DATA_BLOCK "ASW_GraphicData"	// DB 80
TITLE = COPYRIGHT:    (C) 2003  BUHLER AG, CH-9240 UZWIL, SWITZERLAND
//
//PRODUCT:      GP_GCS7
//
//TITLE:        
//
//------------------------------------------------------------------------------------------------------
//
//IDENT:               AUTHOR:         DEPT:                 DATE:
//
//DB80.1A            CE                    FU53                    03.03.2003
//
//------------------------------------------------------------------------------------------------------
//
//PURPOSE:      MANUAL : see [MxxMAN]
//
//RESTRICTIONS: 
//------------------------------------------------------------------------------------------------------
//
//
//
//
AUTHOR : CE
FAMILY : GEN
VERSION : 0.0
  STRUCT
   spare0 : WORD ;
   Buttons : STRUCT
    Fault_F : UDT 1000;	//Fault_F1...Fault_F10
    Fault_SF : UDT 1000;	//Fault_SF1...Fault_SF10
    Active_F : UDT 1000;	//Active_F1...Active_F10
    Active_SF : UDT 1000;	//Active_SF1...Active_SF10
    Manual_F : UDT 1000;	//Manual_F1...Manual_F10
    Manual_SF : UDT 1000;	//Manual_SF1...Manual_SF10
   END_STRUCT ;
   spare14 : ARRAY  [14 .. 29 ] OF BYTE ;
   Way : STRUCT
    F01 : UDT 1001;	//F01L00 ... F01L09
    F02 : UDT 1001;	//F02L00 ... F02L09
    F03 : UDT 1001;	//F03L00 ... F03L09
    F04 : UDT 1001;	//F04L00 ... F04L09
    F05 : UDT 1001;	//F05L00 ... F05L09
    F06 : UDT 1001;	//F06L00 ... F06L09
    F07 : UDT 1001;	//F07L00 ... F07L09
    F08 : UDT 1001;	//F08L00 ... F08L09
    F09 : UDT 1001;	//F09L00 ... F09L09
    F10 : UDT 1001;	//F10L00 ... F10L09
    SF01 : UDT 1001;	//SF01L00 ... SF01L09
    SF02 : UDT 1001;	//SF02L00 ... SF02L09
    SF03 : UDT 1001;	//SF03L00 ... SF03L09
    SF04 : UDT 1001;	//SF04L00 ... SF04L09
    SF05 : UDT 1001;	//SF05L00 ... SF05L09
    SF06 : UDT 1001;	//SF06L00 ... SF06L09
    SF07 : UDT 1001;	//SF07L00 ... SF07L09
    SF08 : UDT 1001;	//SF08L00 ... SF08L09
    SF09 : UDT 1001;	//SF09L00 ... SF09L09
    SF10 : UDT 1001;	//SF10L00 ... SF10L09
   END_STRUCT ;
   Spare430 : ARRAY  [430 .. 499 ] OF BYTE ;
   General : STRUCT
    EmergencyStop : STRUCT
     SystemReset : BOOL ;	//Reset Emergency System
    END_STRUCT ;
    Horn : STRUCT
     Quit : ARRAY  [1 .. 16 ] OF //SwitchOff Horn 1..16
     BOOL ;
     Color : ARRAY  [1 .. 16 ] OF //Horn 1..16 is on
     BOOL ;
    END_STRUCT ;
    CycleTime : ARRAY  [1 .. 3 ] OF //Cycle Time Cycle 1..3
    STRUCT
     Minimal : INT ;	//Min. Cycle Time
     Actual : INT ;	//Act. Cycle Time
     Maximal : INT ;	//Max. Cycle Time
    END_STRUCT ;
    PCS : STRUCT
     PICNotOnline : BOOL ;	//ProcessControlSystem is not online
     Reserve : BOOL ;
    END_STRUCT ;
    Spare526 : STRUCT
     Reserve : ARRAY  [526 .. 549 ] OF BYTE ;
    END_STRUCT ;
   END_STRUCT ;
   UserPictureData : STRUCT
    F1 : STRUCT 	//User Data in Picture F1
     Binaer1 : STRUCT
      Bit0 : BOOL ;
      Bit01 : BOOL ;
      Bit02 : BOOL ;
     END_STRUCT ;
     Binaer2 : STRUCT
      Bit0 : BOOL ;
      Bit01 : BOOL ;
      Bit02 : BOOL ;
     END_STRUCT ;
     Binaer3 : STRUCT
      Bit0 : BOOL ;
      Bit01 : BOOL ;
     END_STRUCT ;
     Binaer4 : STRUCT
      Bit0 : BOOL ;
      Bit01 : BOOL ;
     END_STRUCT ;
     Binaer5 : STRUCT
      Bit0 : BOOL ;
      Bit01 : BOOL ;
     END_STRUCT ;
     Value1 : WORD ;
     Value2 : WORD ;
     Value3 : WORD ;
     Value4 : WORD ;
     Value5 : WORD ;
     Value6 : WORD ;
     Value7 : WORD ;
     Value8 : WORD ;
     Value9 : WORD ;
     Value10 : WORD ;
     Value11 : WORD ;
     Value12 : WORD ;
     Value13 : WORD ;
     Value14 : WORD ;
     Value15 : WORD ;
    END_STRUCT ;
    F2 : STRUCT 	//User Data in Picture F2
     Binaer1 : STRUCT
      Bit0 : BOOL ;
      Bit01 : BOOL ;
      Bit02 : BOOL ;
     END_STRUCT ;
     Binaer2 : STRUCT
      Bit0 : BOOL ;
      Bit01 : BOOL ;
      Bit02 : BOOL ;
     END_STRUCT ;
     Binaer3 : STRUCT
      Bit0 : BOOL ;
      Bit01 : BOOL ;
     END_STRUCT ;
     Binaer4 : STRUCT
      Bit0 : BOOL ;
      Bit01 : BOOL ;
     END_STRUCT ;
     Binaer5 : STRUCT
      Bit0 : BOOL ;
      Bit01 : BOOL ;
     END_STRUCT ;
     Value1 : WORD ;
     Value2 : WORD ;
     Value3 : WORD ;
     Value4 : WORD ;
     Value5 : WORD ;
     Value6 : WORD ;
     Value7 : WORD ;
     Value8 : WORD ;
     Value9 : WORD ;
     Value10 : WORD ;
     Value11 : WORD ;
     Value12 : WORD ;
     Value13 : WORD ;
     Value14 : WORD ;
     Value15 : WORD ;
    END_STRUCT ;
    F3 : STRUCT 	//User Data in Picture F3
     Binaer1 : STRUCT
      Bit0 : BOOL ;
      Bit01 : BOOL ;
      Bit02 : BOOL ;
     END_STRUCT ;
     Binaer2 : STRUCT
      Bit0 : BOOL ;
      Bit01 : BOOL ;
      Bit02 : BOOL ;
     END_STRUCT ;
     Binaer3 : STRUCT
      Bit0 : BOOL ;
      Bit01 : BOOL ;
     END_STRUCT ;
     Binaer4 : STRUCT
      Bit0 : BOOL ;
      Bit01 : BOOL ;
     END_STRUCT ;
     Binaer5 : STRUCT
      Bit0 : BOOL ;
      Bit01 : BOOL ;
     END_STRUCT ;
     Value1 : WORD ;
     Value2 : WORD ;
     Value3 : WORD ;
     Value4 : WORD ;
     Value5 : WORD ;
     Value6 : WORD ;
     Value7 : WORD ;
     Value8 : WORD ;
     Value9 : WORD ;
     Value10 : WORD ;
     Value11 : WORD ;
     Value12 : WORD ;
     Value13 : WORD ;
     Value14 : WORD ;
     Value15 : WORD ;
    END_STRUCT ;
    F4 : STRUCT 	//User Data in Picture F4
     Binaer1 : STRUCT
      Bit0 : BOOL ;
      Bit01 : BOOL ;
      Bit02 : BOOL ;
     END_STRUCT ;
     Binaer2 : STRUCT
      Bit0 : BOOL ;
      Bit01 : BOOL ;
      Bit02 : BOOL ;
     END_STRUCT ;
     Binaer3 : STRUCT
      Bit0 : BOOL ;
      Bit01 : BOOL ;
     END_STRUCT ;
     Binaer4 : STRUCT
      Bit0 : BOOL ;
      Bit01 : BOOL ;
     END_STRUCT ;
     Binaer5 : STRUCT
      Bit0 : BOOL ;
      Bit01 : BOOL ;
     END_STRUCT ;
     Value1 : WORD ;
     Value2 : WORD ;
     Value3 : WORD ;
     Value4 : WORD ;
     Value5 : WORD ;
     Value6 : WORD ;
     Value7 : WORD ;
     Value8 : WORD ;
     Value9 : WORD ;
     Value10 : WORD ;
     Value11 : WORD ;
     Value12 : WORD ;
     Value13 : WORD ;
     Value14 : WORD ;
     Value15 : WORD ;
    END_STRUCT ;
    F5 : STRUCT 	//User Data in Picture F5
     Binaer1 : STRUCT
      Bit0 : BOOL ;
      Bit01 : BOOL ;
      Bit02 : BOOL ;
     END_STRUCT ;
     Binaer2 : STRUCT
      Bit0 : BOOL ;
      Bit01 : BOOL ;
      Bit02 : BOOL ;
     END_STRUCT ;
     Binaer3 : STRUCT
      Bit0 : BOOL ;
      Bit01 : BOOL ;
     END_STRUCT ;
     Binaer4 : STRUCT
      Bit0 : BOOL ;
      Bit01 : BOOL ;
     END_STRUCT ;
     Binaer5 : STRUCT
      Bit0 : BOOL ;
      Bit01 : BOOL ;
     END_STRUCT ;
     Value1 : WORD ;
     Value2 : WORD ;
     Value3 : WORD ;
     Value4 : WORD ;
     Value5 : WORD ;
     Value6 : WORD ;
     Value7 : WORD ;
     Value8 : WORD ;
     Value9 : WORD ;
     Value10 : WORD ;
     Value11 : WORD ;
     Value12 : WORD ;
     Value13 : WORD ;
     Value14 : WORD ;
     Value15 : WORD ;
    END_STRUCT ;
    F6 : STRUCT 	//User Data in Picture F6
     Binaer1 : STRUCT
      Bit0 : BOOL ;
      Bit01 : BOOL ;
      Bit02 : BOOL ;
     END_STRUCT ;
     Binaer2 : STRUCT
      Bit0 : BOOL ;
      Bit01 : BOOL ;
      Bit02 : BOOL ;
     END_STRUCT ;
     Binaer3 : STRUCT
      Bit0 : BOOL ;
      Bit01 : BOOL ;
     END_STRUCT ;
     Binaer4 : STRUCT
      Bit0 : BOOL ;
      Bit01 : BOOL ;
     END_STRUCT ;
     Binaer5 : STRUCT
      Bit0 : BOOL ;
      Bit01 : BOOL ;
     END_STRUCT ;
     Value1 : WORD ;
     Value2 : WORD ;
     Value3 : WORD ;
     Value4 : WORD ;
     Value5 : WORD ;
     Value6 : WORD ;
     Value7 : WORD ;
     Value8 : WORD ;
     Value9 : WORD ;
     Value10 : WORD ;
     Value11 : WORD ;
     Value12 : WORD ;
     Value13 : WORD ;
     Value14 : WORD ;
     Value15 : WORD ;
    END_STRUCT ;
    F7 : STRUCT 	//User Data in Picture F7
     Binaer1 : STRUCT
      Bit0 : BOOL ;
      Bit01 : BOOL ;
      Bit02 : BOOL ;
     END_STRUCT ;
     Binaer2 : STRUCT
      Bit0 : BOOL ;
      Bit01 : BOOL ;
      Bit02 : BOOL ;
     END_STRUCT ;
     Binaer3 : STRUCT
      Bit0 : BOOL ;
      Bit01 : BOOL ;
     END_STRUCT ;
     Binaer4 : STRUCT
      Bit0 : BOOL ;
      Bit01 : BOOL ;
     END_STRUCT ;
     Binaer5 : STRUCT
      Bit0 : BOOL ;
      Bit01 : BOOL ;
     END_STRUCT ;
     Value1 : WORD ;
     Value2 : WORD ;
     Value3 : WORD ;
     Value4 : WORD ;
     Value5 : WORD ;
     Value6 : WORD ;
     Value7 : WORD ;
     Value8 : WORD ;
     Value9 : WORD ;
     Value10 : WORD ;
     Value11 : WORD ;
     Value12 : WORD ;
     Value13 : WORD ;
     Value14 : WORD ;
     Value15 : WORD ;
    END_STRUCT ;
    F8 : STRUCT 	//User Data in Picture F8
     Binaer1 : STRUCT
      Bit0 : BOOL ;
      Bit01 : BOOL ;
      Bit02 : BOOL ;
     END_STRUCT ;
     Binaer2 : STRUCT
      Bit0 : BOOL ;
      Bit01 : BOOL ;
      Bit02 : BOOL ;
     END_STRUCT ;
     Binaer3 : STRUCT
      Bit0 : BOOL ;
      Bit01 : BOOL ;
     END_STRUCT ;
     Binaer4 : STRUCT
      Bit0 : BOOL ;
      Bit01 : BOOL ;
     END_STRUCT ;
     Binaer5 : STRUCT
      Bit0 : BOOL ;
      Bit01 : BOOL ;
     END_STRUCT ;
     Value1 : WORD ;
     Value2 : WORD ;
     Value3 : WORD ;
     Value4 : WORD ;
     Value5 : WORD ;
     Value6 : WORD ;
     Value7 : WORD ;
     Value8 : WORD ;
     Value9 : WORD ;
     Value10 : WORD ;
     Value11 : WORD ;
     Value12 : WORD ;
     Value13 : WORD ;
     Value14 : WORD ;
     Value15 : WORD ;
    END_STRUCT ;
    F9 : STRUCT 	//User Data in Picture F9
     Binaer1 : STRUCT
      Bit0 : BOOL ;
      Bit01 : BOOL ;
      Bit02 : BOOL ;
     END_STRUCT ;
     Binaer2 : STRUCT
      Bit0 : BOOL ;
      Bit01 : BOOL ;
      Bit02 : BOOL ;
     END_STRUCT ;
     Binaer3 : STRUCT
      Bit0 : BOOL ;
      Bit01 : BOOL ;
     END_STRUCT ;
     Binaer4 : STRUCT
      Bit0 : BOOL ;
      Bit01 : BOOL ;
     END_STRUCT ;
     Binaer5 : STRUCT
      Bit0 : BOOL ;
      Bit01 : BOOL ;
     END_STRUCT ;
     Value1 : WORD ;
     Value2 : WORD ;
     Value3 : WORD ;
     Value4 : WORD ;
     Value5 : WORD ;
     Value6 : WORD ;
     Value7 : WORD ;
     Value8 : WORD ;
     Value9 : WORD ;
     Value10 : WORD ;
     Value11 : WORD ;
     Value12 : WORD ;
     Value13 : WORD ;
     Value14 : WORD ;
     Value15 : WORD ;
    END_STRUCT ;
    F10 : STRUCT 	//User Data in Picture F10
     Binaer1 : STRUCT
      Bit0 : BOOL ;
      Bit01 : BOOL ;
      Bit02 : BOOL ;
     END_STRUCT ;
     Binaer2 : STRUCT
      Bit0 : BOOL ;
      Bit01 : BOOL ;
      Bit02 : BOOL ;
     END_STRUCT ;
     Binaer3 : STRUCT
      Bit0 : BOOL ;
      Bit01 : BOOL ;
     END_STRUCT ;
     Binaer4 : STRUCT
      Bit0 : BOOL ;
      Bit01 : BOOL ;
     END_STRUCT ;
     Binaer5 : STRUCT
      Bit0 : BOOL ;
      Bit01 : BOOL ;
     END_STRUCT ;
     Value1 : WORD ;
     Value2 : WORD ;
     Value3 : WORD ;
     Value4 : WORD ;
     Value5 : WORD ;
     Value6 : WORD ;
     Value7 : WORD ;
     Value8 : WORD ;
     Value9 : WORD ;
     Value10 : WORD ;
     Value11 : WORD ;
     Value12 : WORD ;
     Value13 : WORD ;
     Value14 : WORD ;
     Value15 : WORD ;
    END_STRUCT ;
    SF1 : STRUCT 	//User Data in Picture SF1
     Binaer1 : STRUCT
      Bit0 : BOOL ;
      Bit01 : BOOL ;
      Bit02 : BOOL ;
     END_STRUCT ;
     Binaer2 : STRUCT
      Bit0 : BOOL ;
      Bit01 : BOOL ;
      Bit02 : BOOL ;
     END_STRUCT ;
     Binaer3 : STRUCT
      Bit0 : BOOL ;
      Bit01 : BOOL ;
     END_STRUCT ;
     Binaer4 : STRUCT
      Bit0 : BOOL ;
      Bit01 : BOOL ;
     END_STRUCT ;
     Binaer5 : STRUCT
      Bit0 : BOOL ;
      Bit01 : BOOL ;
     END_STRUCT ;
     Value1 : WORD ;
     Value2 : WORD ;
     Value3 : WORD ;
     Value4 : WORD ;
     Value5 : WORD ;
     Value6 : WORD ;
     Value7 : WORD ;
     Value8 : WORD ;
     Value9 : WORD ;
     Value10 : WORD ;
     Value11 : WORD ;
     Value12 : WORD ;
     Value13 : WORD ;
     Value14 : WORD ;
     Value15 : WORD ;
    END_STRUCT ;
    SF2 : STRUCT 	//User Data in Picture SF2
     Binaer1 : STRUCT
      Bit0 : BOOL ;
      Bit01 : BOOL ;
      Bit02 : BOOL ;
     END_STRUCT ;
     Binaer2 : STRUCT
      Bit0 : BOOL ;
      Bit01 : BOOL ;
      Bit02 : BOOL ;
     END_STRUCT ;
     Binaer3 : STRUCT
      Bit0 : BOOL ;
      Bit01 : BOOL ;
     END_STRUCT ;
     Binaer4 : STRUCT
      Bit0 : BOOL ;
      Bit01 : BOOL ;
     END_STRUCT ;
     Binaer5 : STRUCT
      Bit0 : BOOL ;
      Bit01 : BOOL ;
     END_STRUCT ;
     Value1 : WORD ;
     Value2 : WORD ;
     Value3 : WORD ;
     Value4 : WORD ;
     Value5 : WORD ;
     Value6 : WORD ;
     Value7 : WORD ;
     Value8 : WORD ;
     Value9 : WORD ;
     Value10 : WORD ;
     Value11 : WORD ;
     Value12 : WORD ;
     Value13 : WORD ;
     Value14 : WORD ;
     Value15 : WORD ;
    END_STRUCT ;
    SF3 : STRUCT 	//User Data in Picture SF3
     Binaer1 : STRUCT
      Bit0 : BOOL ;
      Bit01 : BOOL ;
      Bit02 : BOOL ;
     END_STRUCT ;
     Binaer2 : STRUCT
      Bit0 : BOOL ;
      Bit01 : BOOL ;
      Bit02 : BOOL ;
     END_STRUCT ;
     Binaer3 : STRUCT
      Bit0 : BOOL ;
      Bit01 : BOOL ;
     END_STRUCT ;
     Binaer4 : STRUCT
      Bit0 : BOOL ;
      Bit01 : BOOL ;
     END_STRUCT ;
     Binaer5 : STRUCT
      Bit0 : BOOL ;
      Bit01 : BOOL ;
     END_STRUCT ;
     Value1 : WORD ;
     Value2 : WORD ;
     Value3 : WORD ;
     Value4 : WORD ;
     Value5 : WORD ;
     Value6 : WORD ;
     Value7 : WORD ;
     Value8 : WORD ;
     Value9 : WORD ;
     Value10 : WORD ;
     Value11 : WORD ;
     Value12 : WORD ;
     Value13 : WORD ;
     Value14 : WORD ;
     Value15 : WORD ;
    END_STRUCT ;
    SF4 : STRUCT 	//User Data in Picture SF4
     Binaer1 : STRUCT
      Bit0 : BOOL ;
      Bit01 : BOOL ;
      Bit02 : BOOL ;
     END_STRUCT ;
     Binaer2 : STRUCT
      Bit0 : BOOL ;
      Bit01 : BOOL ;
      Bit02 : BOOL ;
     END_STRUCT ;
     Binaer3 : STRUCT
      Bit0 : BOOL ;
      Bit01 : BOOL ;
     END_STRUCT ;
     Binaer4 : STRUCT
      Bit0 : BOOL ;
      Bit01 : BOOL ;
     END_STRUCT ;
     Binaer5 : STRUCT
      Bit0 : BOOL ;
      Bit01 : BOOL ;
     END_STRUCT ;
     Value1 : WORD ;
     Value2 : WORD ;
     Value3 : WORD ;
     Value4 : WORD ;
     Value5 : WORD ;
     Value6 : WORD ;
     Value7 : WORD ;
     Value8 : WORD ;
     Value9 : WORD ;
     Value10 : WORD ;
     Value11 : WORD ;
     Value12 : WORD ;
     Value13 : WORD ;
     Value14 : WORD ;
     Value15 : WORD ;
    END_STRUCT ;
    SF5 : STRUCT 	//User Data in Picture SF5
     Binaer1 : STRUCT
      Bit0 : BOOL ;
      Bit01 : BOOL ;
      Bit02 : BOOL ;
     END_STRUCT ;
     Binaer2 : STRUCT
      Bit0 : BOOL ;
      Bit01 : BOOL ;
      Bit02 : BOOL ;
     END_STRUCT ;
     Binaer3 : STRUCT
      Bit0 : BOOL ;
      Bit01 : BOOL ;
     END_STRUCT ;
     Binaer4 : STRUCT
      Bit0 : BOOL ;
      Bit01 : BOOL ;
     END_STRUCT ;
     Binaer5 : STRUCT
      Bit0 : BOOL ;
      Bit01 : BOOL ;
     END_STRUCT ;
     Value1 : WORD ;
     Value2 : WORD ;
     Value3 : WORD ;
     Value4 : WORD ;
     Value5 : WORD ;
     Value6 : WORD ;
     Value7 : WORD ;
     Value8 : WORD ;
     Value9 : WORD ;
     Value10 : WORD ;
     Value11 : WORD ;
     Value12 : WORD ;
     Value13 : WORD ;
     Value14 : WORD ;
     Value15 : WORD ;
    END_STRUCT ;
    SF6 : STRUCT 	//User Data in Picture SF6
     Binaer1 : STRUCT
      Bit0 : BOOL ;
      Bit01 : BOOL ;
      Bit02 : BOOL ;
     END_STRUCT ;
     Binaer2 : STRUCT
      Bit0 : BOOL ;
      Bit01 : BOOL ;
      Bit02 : BOOL ;
     END_STRUCT ;
     Binaer3 : STRUCT
      Bit0 : BOOL ;
      Bit01 : BOOL ;
     END_STRUCT ;
     Binaer4 : STRUCT
      Bit0 : BOOL ;
      Bit01 : BOOL ;
     END_STRUCT ;
     Binaer5 : STRUCT
      Bit0 : BOOL ;
      Bit01 : BOOL ;
     END_STRUCT ;
     Value1 : WORD ;
     Value2 : WORD ;
     Value3 : WORD ;
     Value4 : WORD ;
     Value5 : WORD ;
     Value6 : WORD ;
     Value7 : WORD ;
     Value8 : WORD ;
     Value9 : WORD ;
     Value10 : WORD ;
     Value11 : WORD ;
     Value12 : WORD ;
     Value13 : WORD ;
     Value14 : WORD ;
     Value15 : WORD ;
    END_STRUCT ;
    SF7 : STRUCT 	//User Data in Picture SF7
     Binaer1 : STRUCT
      Bit0 : BOOL ;
      Bit01 : BOOL ;
      Bit02 : BOOL ;
     END_STRUCT ;
     Binaer2 : STRUCT
      Bit0 : BOOL ;
      Bit01 : BOOL ;
      Bit02 : BOOL ;
     END_STRUCT ;
     Binaer3 : STRUCT
      Bit0 : BOOL ;
      Bit01 : BOOL ;
     END_STRUCT ;
     Binaer4 : STRUCT
      Bit0 : BOOL ;
      Bit01 : BOOL ;
     END_STRUCT ;
     Binaer5 : STRUCT
      Bit0 : BOOL ;
      Bit01 : BOOL ;
     END_STRUCT ;
     Value1 : WORD ;
     Value2 : WORD ;
     Value3 : WORD ;
     Value4 : WORD ;
     Value5 : WORD ;
     Value6 : WORD ;
     Value7 : WORD ;
     Value8 : WORD ;
     Value9 : WORD ;
     Value10 : WORD ;
     Value11 : WORD ;
     Value12 : WORD ;
     Value13 : WORD ;
     Value14 : WORD ;
     Value15 : WORD ;
    END_STRUCT ;
    SF8 : STRUCT 	//User Data in Picture SF8
     Binaer1 : STRUCT
      Bit0 : BOOL ;
      Bit01 : BOOL ;
      Bit02 : BOOL ;
     END_STRUCT ;
     Binaer2 : STRUCT
      Bit0 : BOOL ;
      Bit01 : BOOL ;
      Bit02 : BOOL ;
     END_STRUCT ;
     Binaer3 : STRUCT
      Bit0 : BOOL ;
      Bit01 : BOOL ;
     END_STRUCT ;
     Binaer4 : STRUCT
      Bit0 : BOOL ;
      Bit01 : BOOL ;
     END_STRUCT ;
     Binaer5 : STRUCT
      Bit0 : BOOL ;
      Bit01 : BOOL ;
     END_STRUCT ;
     Value1 : WORD ;
     Value2 : WORD ;
     Value3 : WORD ;
     Value4 : WORD ;
     Value5 : WORD ;
     Value6 : WORD ;
     Value7 : WORD ;
     Value8 : WORD ;
     Value9 : WORD ;
     Value10 : WORD ;
     Value11 : WORD ;
     Value12 : WORD ;
     Value13 : WORD ;
     Value14 : WORD ;
     Value15 : WORD ;
    END_STRUCT ;
    SF9 : STRUCT 	//User Data in Picture SF9
     Binaer1 : STRUCT
      Bit0 : BOOL ;
      Bit01 : BOOL ;
      Bit02 : BOOL ;
     END_STRUCT ;
     Binaer2 : STRUCT
      Bit0 : BOOL ;
      Bit01 : BOOL ;
      Bit02 : BOOL ;
     END_STRUCT ;
     Binaer3 : STRUCT
      Bit0 : BOOL ;
      Bit01 : BOOL ;
     END_STRUCT ;
     Binaer4 : STRUCT
      Bit0 : BOOL ;
      Bit01 : BOOL ;
     END_STRUCT ;
     Binaer5 : STRUCT
      Bit0 : BOOL ;
      Bit01 : BOOL ;
     END_STRUCT ;
     Value1 : WORD ;
     Value2 : WORD ;
     Value3 : WORD ;
     Value4 : WORD ;
     Value5 : WORD ;
     Value6 : WORD ;
     Value7 : WORD ;
     Value8 : WORD ;
     Value9 : WORD ;
     Value10 : WORD ;
     Value11 : WORD ;
     Value12 : WORD ;
     Value13 : WORD ;
     Value14 : WORD ;
     Value15 : WORD ;
    END_STRUCT ;
    SF10 : STRUCT 	//User Data in Picture SF10
     Binaer1 : STRUCT
      Bit0 : BOOL ;
      Bit01 : BOOL ;
      Bit02 : BOOL ;
     END_STRUCT ;
     Binaer2 : STRUCT
      Bit0 : BOOL ;
      Bit01 : BOOL ;
      Bit02 : BOOL ;
     END_STRUCT ;
     Binaer3 : STRUCT
      Bit0 : BOOL ;
      Bit01 : BOOL ;
     END_STRUCT ;
     Binaer4 : STRUCT
      Bit0 : BOOL ;
      Bit01 : BOOL ;
     END_STRUCT ;
     Binaer5 : STRUCT
      Bit0 : BOOL ;
      Bit01 : BOOL ;
     END_STRUCT ;
     Value1 : WORD ;
     Value2 : WORD ;
     Value3 : WORD ;
     Value4 : WORD ;
     Value5 : WORD ;
     Value6 : WORD ;
     Value7 : WORD ;
     Value8 : WORD ;
     Value9 : WORD ;
     Value10 : WORD ;
     Value11 : WORD ;
     Value12 : WORD ;
     Value13 : WORD ;
     Value14 : WORD ;
     Value15 : WORD ;
    END_STRUCT ;
    General : STRUCT 	//User Data in Picture General
     Binaer1 : STRUCT
      Bit0 : BOOL ;
      Bit01 : BOOL ;
      Bit02 : BOOL ;
     END_STRUCT ;
     Binaer2 : STRUCT
      Bit0 : BOOL ;
      Bit01 : BOOL ;
      Bit02 : BOOL ;
     END_STRUCT ;
     Binaer3 : STRUCT
      Bit0 : BOOL ;
      Bit01 : BOOL ;
     END_STRUCT ;
     Binaer4 : STRUCT
      Bit0 : BOOL ;
      Bit01 : BOOL ;
     END_STRUCT ;
     Binaer5 : STRUCT
      Bit0 : BOOL ;
      Bit01 : BOOL ;
     END_STRUCT ;
     Value1 : WORD ;
     Value2 : WORD ;
     Value3 : WORD ;
     Value4 : WORD ;
     Value5 : WORD ;
     Value6 : WORD ;
     Value7 : WORD ;
     Value8 : WORD ;
     Value9 : WORD ;
     Value10 : WORD ;
     Value11 : WORD ;
     Value12 : WORD ;
     Value13 : WORD ;
     Value14 : WORD ;
     Value15 : WORD ;
    END_STRUCT ;
    Liquid : STRUCT 	//User Data in Picture Liquid
     Binaer1 : STRUCT
      Bit0 : BOOL ;
      Bit01 : BOOL ;
      Bit02 : BOOL ;
     END_STRUCT ;
     Binaer2 : STRUCT
      Bit0 : BOOL ;
      Bit01 : BOOL ;
      Bit02 : BOOL ;
     END_STRUCT ;
     Binaer3 : STRUCT
      Bit0 : BOOL ;
      Bit01 : BOOL ;
     END_STRUCT ;
     Binaer4 : STRUCT
      Bit0 : BOOL ;
      Bit01 : BOOL ;
     END_STRUCT ;
     Binaer5 : STRUCT
      Bit0 : BOOL ;
      Bit01 : BOOL ;
     END_STRUCT ;
     Value1 : WORD ;
     Value2 : WORD ;
     Value3 : WORD ;
     Value4 : WORD ;
     Value5 : WORD ;
     Value6 : WORD ;
     Value7 : WORD ;
     Value8 : WORD ;
     Value9 : WORD ;
     Value10 : WORD ;
     Value11 : WORD ;
     Value12 : WORD ;
     Value13 : WORD ;
     Value14 : WORD ;
     Value15 : WORD ;
    END_STRUCT ;
    Spare : STRUCT 	//User Data in Picture Spare
     Binaer1 : STRUCT
      Bit0 : BOOL ;
      Bit01 : BOOL ;
      Bit02 : BOOL ;
     END_STRUCT ;
     Binaer2 : STRUCT
      Bit0 : BOOL ;
      Bit01 : BOOL ;
      Bit02 : BOOL ;
     END_STRUCT ;
     Binaer3 : STRUCT
      Bit0 : BOOL ;
      Bit01 : BOOL ;
     END_STRUCT ;
     Binaer4 : STRUCT
      Bit0 : BOOL ;
      Bit01 : BOOL ;
     END_STRUCT ;
     Binaer5 : STRUCT
      Bit0 : BOOL ;
      Bit01 : BOOL ;
     END_STRUCT ;
     Value1 : WORD ;
     Value2 : WORD ;
     Value3 : WORD ;
     Value4 : WORD ;
     Value5 : WORD ;
     Value6 : WORD ;
     Value7 : WORD ;
     Value8 : WORD ;
     Value9 : WORD ;
     Value10 : WORD ;
     Value11 : WORD ;
     Value12 : WORD ;
     Value13 : WORD ;
     Value14 : WORD ;
     Value15 : WORD ;
    END_STRUCT ;
   END_STRUCT ;
   Spare1470 : STRUCT
    Reserve : ARRAY  [1470 .. 1499 ] OF BYTE ;
   END_STRUCT ;
   GraficDisplayData : STRUCT
    Value1 : DINT ;
    Value2 : DINT ;
    Value3 : DINT ;
    Value4 : DINT ;
    Value5 : DINT ;
    Value6 : DINT ;
    Value7 : DINT ;
    Value8 : DINT ;
    Value9 : DINT ;
    Value10 : DINT ;
    Value11 : DINT ;
    Value12 : DINT ;
    Value13 : DINT ;
    Value14 : DINT ;
    Value15 : DINT ;
    Value16 : DINT ;
    Value17 : DINT ;
    Value18 : DINT ;
    Value19 : DINT ;
    Value20 : DINT ;
    Value21 : DINT ;
    Value22 : DINT ;
    Value23 : DINT ;
    Value24 : DINT ;
    Value25 : DINT ;
    Value26 : DINT ;
    Value27 : DINT ;
    Value28 : DINT ;
    Value29 : DINT ;
    Value30 : DINT ;
    Value31 : DINT ;
    Value32 : DINT ;
    Value33 : DINT ;
    Value34 : DINT ;
    Value35 : DINT ;
    Value36 : DINT ;
    Value37 : DINT ;
    Value38 : DINT ;
    Value39 : DINT ;
    Value40 : DINT ;
    Value41 : DINT ;
    Value42 : DINT ;
    Value43 : DINT ;
    Value44 : DINT ;
    Value45 : DINT ;
    Value46 : DINT ;
    Value47 : DINT ;
    Value48 : DINT ;
    Value49 : DINT ;
    Value50 : DINT ;
    Value51 : DINT ;
    Value52 : DINT ;
    Value53 : DINT ;
    Value54 : DINT ;
    Value55 : DINT ;
    Value56 : DINT ;
    Value57 : DINT ;
    Value58 : DINT ;
    Value59 : DINT ;
    Value60 : DINT ;
    Value61 : DINT ;
    Value62 : DINT ;
    Value63 : DINT ;
    Value64 : DINT ;
    Value65 : DINT ;
    Value66 : DINT ;
    Value67 : DINT ;
    Value68 : DINT ;
    Value69 : DINT ;
    Value70 : DINT ;
    Value71 : DINT ;
    Value72 : DINT ;
    Value73 : DINT ;
    Value74 : DINT ;
    Value75 : DINT ;
    Value76 : DINT ;
    Value77 : DINT ;
    Value78 : DINT ;
    Value79 : DINT ;
    Value80 : DINT ;
    Value81 : DINT ;
    Value82 : DINT ;
    Value83 : DINT ;
    Value84 : DINT ;
    Value85 : DINT ;
    Value86 : DINT ;
    Value87 : DINT ;
    Value88 : DINT ;
    Value89 : DINT ;
    Value90 : DINT ;
    Value91 : DINT ;
    Value92 : DINT ;
    Value93 : DINT ;
    Value94 : DINT ;
    Value95 : DINT ;
    Value96 : DINT ;
    Value97 : DINT ;
    Value98 : DINT ;
    Value99 : DINT ;
    Boolean : STRUCT
     Signal25 : BOOL ;
     Signal26 : BOOL ;
     Signal27 : BOOL ;
     Signal28 : BOOL ;
     Signal29 : BOOL ;
     Signal30 : BOOL ;
     Signal31 : BOOL ;
     Signal32 : BOOL ;
     Signal17 : BOOL ;
     Signal18 : BOOL ;
     Signal19 : BOOL ;
     Signal20 : BOOL ;
     Signal21 : BOOL ;
     Signal22 : BOOL ;
     Signal23 : BOOL ;
     Signal24 : BOOL ;
     Signal09 : BOOL ;
     Signal10 : BOOL ;
     Signal11 : BOOL ;
     Signal12 : BOOL ;
     Signal13 : BOOL ;
     Signal14 : BOOL ;
     Signal15 : BOOL ;
     Signal16 : BOOL ;
     Signal01 : BOOL ;
     Signal02 : BOOL ;
     Signal03 : BOOL ;
     Signal04 : BOOL ;
     Signal05 : BOOL ;
     Signal06 : BOOL ;
     Signal07 : BOOL ;
     Signal08 : BOOL ;
    END_STRUCT ;
   END_STRUCT ;
  END_STRUCT ;	
BEGIN
END_DATA_BLOCK

DATA_BLOCK "ASW_LineInfoData"	// DB 82
TITLE = COPYRIGHT:    (C) 2003  BUHLER AG, CH-9240 UZWIL, SWITZERLAND
//
//PRODUCT:      GP_GCS7
//
//TITLE:        
//
//------------------------------------------------------------------------------------------------------
//
//IDENT:               AUTHOR:         DEPT:                 DATE:
//
//DB82.1A            CE                    FU53                    03.03.2003
//
//------------------------------------------------------------------------------------------------------
//
//PURPOSE:      MANUAL : see [MxxMAN]
//
//RESTRICTIONS: 
//------------------------------------------------------------------------------------------------------
//
//
//
//
//
AUTHOR : CE
FAMILY : USW
VERSION : 0.0
  STRUCT
   Reserve0 : ARRAY  [0 .. 99 ] OF BYTE ;
   MIX_LINE : ARRAY  [1 .. 10 ] OF UDT 1003;
   TRSP_LINE : ARRAY  [11 .. 32 ] OF UDT 1003;
  END_STRUCT ;	
BEGIN
   MIX_LINE[1].ProductIdent := 'ABCDEFGHIJKLMNOP';
   MIX_LINE[1].ProductName := 'ABCDEFGHIJKLMNOPQRSTUVWXYZ012345';
   MIX_LINE[1].LOT_NR_1 := 'ABCDEFGHIJKLMNOP';
   MIX_LINE[1].LOT_NR_2 := 'ABCDEFGHIJKLMNOP';
   MIX_LINE[1].LOT_NR_3 := 'ABCDEFGHIJKLMNOP';
   MIX_LINE[2].ProductIdent := 'ABCDEFGHIJKLMNOP';
   MIX_LINE[2].ProductName := 'ABCDEFGHIJKLMNOPQRSTUVWXYZ012345';
   MIX_LINE[2].LOT_NR_1 := 'ABCDEFGHIJKLMNOP';
   MIX_LINE[2].LOT_NR_2 := 'ABCDEFGHIJKLMNOP';
   MIX_LINE[2].LOT_NR_3 := 'ABCDEFGHIJKLMNOP';
   MIX_LINE[3].ProductIdent := 'ABCDEFGHIJKLMNOP';
   MIX_LINE[3].ProductName := 'ABCDEFGHIJKLMNOPQRSTUVWXYZ012345';
   MIX_LINE[3].LOT_NR_1 := 'ABCDEFGHIJKLMNOP';
   MIX_LINE[3].LOT_NR_2 := 'ABCDEFGHIJKLMNOP';
   MIX_LINE[3].LOT_NR_3 := 'ABCDEFGHIJKLMNOP';
   MIX_LINE[4].ProductIdent := 'ABCDEFGHIJKLMNOP';
   MIX_LINE[4].ProductName := 'ABCDEFGHIJKLMNOPQRSTUVWXYZ012345';
   MIX_LINE[4].LOT_NR_1 := 'ABCDEFGHIJKLMNOP';
   MIX_LINE[4].LOT_NR_2 := 'ABCDEFGHIJKLMNOP';
   MIX_LINE[4].LOT_NR_3 := 'ABCDEFGHIJKLMNOP';
   MIX_LINE[5].ProductIdent := 'ABCDEFGHIJKLMNOP';
   MIX_LINE[5].ProductName := 'ABCDEFGHIJKLMNOPQRSTUVWXYZ012345';
   MIX_LINE[5].LOT_NR_1 := 'ABCDEFGHIJKLMNOP';
   MIX_LINE[5].LOT_NR_2 := 'ABCDEFGHIJKLMNOP';
   MIX_LINE[5].LOT_NR_3 := 'ABCDEFGHIJKLMNOP';
   MIX_LINE[6].ProductIdent := 'ABCDEFGHIJKLMNOP';
   MIX_LINE[6].ProductName := 'ABCDEFGHIJKLMNOPQRSTUVWXYZ012345';
   MIX_LINE[6].LOT_NR_1 := 'ABCDEFGHIJKLMNOP';
   MIX_LINE[6].LOT_NR_2 := 'ABCDEFGHIJKLMNOP';
   MIX_LINE[6].LOT_NR_3 := 'ABCDEFGHIJKLMNOP';
   MIX_LINE[7].ProductIdent := 'ABCDEFGHIJKLMNOP';
   MIX_LINE[7].ProductName := 'ABCDEFGHIJKLMNOPQRSTUVWXYZ012345';
   MIX_LINE[7].LOT_NR_1 := 'ABCDEFGHIJKLMNOP';
   MIX_LINE[7].LOT_NR_2 := 'ABCDEFGHIJKLMNOP';
   MIX_LINE[7].LOT_NR_3 := 'ABCDEFGHIJKLMNOP';
   MIX_LINE[8].ProductIdent := 'ABCDEFGHIJKLMNOP';
   MIX_LINE[8].ProductName := 'ABCDEFGHIJKLMNOPQRSTUVWXYZ012345';
   MIX_LINE[8].LOT_NR_1 := 'ABCDEFGHIJKLMNOP';
   MIX_LINE[8].LOT_NR_2 := 'ABCDEFGHIJKLMNOP';
   MIX_LINE[8].LOT_NR_3 := 'ABCDEFGHIJKLMNOP';
   MIX_LINE[9].ProductIdent := 'ABCDEFGHIJKLMNOP';
   MIX_LINE[9].ProductName := 'ABCDEFGHIJKLMNOPQRSTUVWXYZ012345';
   MIX_LINE[9].LOT_NR_1 := 'ABCDEFGHIJKLMNOP';
   MIX_LINE[9].LOT_NR_2 := 'ABCDEFGHIJKLMNOP';
   MIX_LINE[9].LOT_NR_3 := 'ABCDEFGHIJKLMNOP';
   MIX_LINE[10].ProductIdent := 'ABCDEFGHIJKLMNOP';
   MIX_LINE[10].ProductName := 'ABCDEFGHIJKLMNOPQRSTUVWXYZ012345';
   MIX_LINE[10].LOT_NR_1 := 'ABCDEFGHIJKLMNOP';
   MIX_LINE[10].LOT_NR_2 := 'ABCDEFGHIJKLMNOP';
   MIX_LINE[10].LOT_NR_3 := 'ABCDEFGHIJKLMNOP';
   TRSP_LINE[11].ProductIdent := 'ABCDEFGHIJKLMNOP';
   TRSP_LINE[11].ProductName := 'ABCDEFGHIJKLMNOPQRSTUVWXYZ012345';
   TRSP_LINE[11].LOT_NR_1 := 'ABCDEFGHIJKLMNOP';
   TRSP_LINE[11].LOT_NR_2 := 'ABCDEFGHIJKLMNOP';
   TRSP_LINE[11].LOT_NR_3 := 'ABCDEFGHIJKLMNOP';
   TRSP_LINE[12].ProductIdent := 'ABCDEFGHIJKLMNOP';
   TRSP_LINE[12].ProductName := 'ABCDEFGHIJKLMNOPQRSTUVWXYZ012345';
   TRSP_LINE[12].LOT_NR_1 := 'ABCDEFGHIJKLMNOP';
   TRSP_LINE[12].LOT_NR_2 := 'ABCDEFGHIJKLMNOP';
   TRSP_LINE[12].LOT_NR_3 := 'ABCDEFGHIJKLMNOP';
   TRSP_LINE[13].ProductIdent := 'ABCDEFGHIJKLMNOP';
   TRSP_LINE[13].ProductName := 'ABCDEFGHIJKLMNOPQRSTUVWXYZ012345';
   TRSP_LINE[13].LOT_NR_1 := 'ABCDEFGHIJKLMNOP';
   TRSP_LINE[13].LOT_NR_2 := 'ABCDEFGHIJKLMNOP';
   TRSP_LINE[13].LOT_NR_3 := 'ABCDEFGHIJKLMNOP';
   TRSP_LINE[14].ProductIdent := 'ABCDEFGHIJKLMNOP';
   TRSP_LINE[14].ProductName := 'ABCDEFGHIJKLMNOPQRSTUVWXYZ012345';
   TRSP_LINE[14].LOT_NR_1 := 'ABCDEFGHIJKLMNOP';
   TRSP_LINE[14].LOT_NR_2 := 'ABCDEFGHIJKLMNOP';
   TRSP_LINE[14].LOT_NR_3 := 'ABCDEFGHIJKLMNOP';
   TRSP_LINE[15].ProductIdent := 'ABCDEFGHIJKLMNOP';
   TRSP_LINE[15].ProductName := 'ABCDEFGHIJKLMNOPQRSTUVWXYZ012345';
   TRSP_LINE[15].LOT_NR_1 := 'ABCDEFGHIJKLMNOP';
   TRSP_LINE[15].LOT_NR_2 := 'ABCDEFGHIJKLMNOP';
   TRSP_LINE[15].LOT_NR_3 := 'ABCDEFGHIJKLMNOP';
   TRSP_LINE[16].ProductIdent := 'ABCDEFGHIJKLMNOP';
   TRSP_LINE[16].ProductName := 'ABCDEFGHIJKLMNOPQRSTUVWXYZ012345';
   TRSP_LINE[16].LOT_NR_1 := 'ABCDEFGHIJKLMNOP';
   TRSP_LINE[16].LOT_NR_2 := 'ABCDEFGHIJKLMNOP';
   TRSP_LINE[16].LOT_NR_3 := 'ABCDEFGHIJKLMNOP';
   TRSP_LINE[17].ProductIdent := 'ABCDEFGHIJKLMNOP';
   TRSP_LINE[17].ProductName := 'ABCDEFGHIJKLMNOPQRSTUVWXYZ012345';
   TRSP_LINE[17].LOT_NR_1 := 'ABCDEFGHIJKLMNOP';
   TRSP_LINE[17].LOT_NR_2 := 'ABCDEFGHIJKLMNOP';
   TRSP_LINE[17].LOT_NR_3 := 'ABCDEFGHIJKLMNOP';
   TRSP_LINE[18].ProductIdent := 'ABCDEFGHIJKLMNOP';
   TRSP_LINE[18].ProductName := 'ABCDEFGHIJKLMNOPQRSTUVWXYZ012345';
   TRSP_LINE[18].LOT_NR_1 := 'ABCDEFGHIJKLMNOP';
   TRSP_LINE[18].LOT_NR_2 := 'ABCDEFGHIJKLMNOP';
   TRSP_LINE[18].LOT_NR_3 := 'ABCDEFGHIJKLMNOP';
   TRSP_LINE[19].ProductIdent := 'ABCDEFGHIJKLMNOP';
   TRSP_LINE[19].ProductName := 'ABCDEFGHIJKLMNOPQRSTUVWXYZ012345';
   TRSP_LINE[19].LOT_NR_1 := 'ABCDEFGHIJKLMNOP';
   TRSP_LINE[19].LOT_NR_2 := 'ABCDEFGHIJKLMNOP';
   TRSP_LINE[19].LOT_NR_3 := 'ABCDEFGHIJKLMNOP';
   TRSP_LINE[20].ProductIdent := 'ABCDEFGHIJKLMNOP';
   TRSP_LINE[20].ProductName := 'ABCDEFGHIJKLMNOPQRSTUVWXYZ012345';
   TRSP_LINE[20].LOT_NR_1 := 'ABCDEFGHIJKLMNOP';
   TRSP_LINE[20].LOT_NR_2 := 'ABCDEFGHIJKLMNOP';
   TRSP_LINE[20].LOT_NR_3 := 'ABCDEFGHIJKLMNOP';
   TRSP_LINE[21].ProductIdent := 'ABCDEFGHIJKLMNOP';
   TRSP_LINE[21].ProductName := 'ABCDEFGHIJKLMNOPQRSTUVWXYZ012345';
   TRSP_LINE[21].LOT_NR_1 := 'ABCDEFGHIJKLMNOP';
   TRSP_LINE[21].LOT_NR_2 := 'ABCDEFGHIJKLMNOP';
   TRSP_LINE[21].LOT_NR_3 := 'ABCDEFGHIJKLMNOP';
   TRSP_LINE[22].ProductIdent := 'ABCDEFGHIJKLMNOP';
   TRSP_LINE[22].ProductName := 'ABCDEFGHIJKLMNOPQRSTUVWXYZ012345';
   TRSP_LINE[22].LOT_NR_1 := 'ABCDEFGHIJKLMNOP';
   TRSP_LINE[22].LOT_NR_2 := 'ABCDEFGHIJKLMNOP';
   TRSP_LINE[22].LOT_NR_3 := 'ABCDEFGHIJKLMNOP';
   TRSP_LINE[23].ProductIdent := 'ABCDEFGHIJKLMNOP';
   TRSP_LINE[23].ProductName := 'ABCDEFGHIJKLMNOPQRSTUVWXYZ012345';
   TRSP_LINE[23].LOT_NR_1 := 'ABCDEFGHIJKLMNOP';
   TRSP_LINE[23].LOT_NR_2 := 'ABCDEFGHIJKLMNOP';
   TRSP_LINE[23].LOT_NR_3 := 'ABCDEFGHIJKLMNOP';
   TRSP_LINE[24].ProductIdent := 'ABCDEFGHIJKLMNOP';
   TRSP_LINE[24].ProductName := 'ABCDEFGHIJKLMNOPQRSTUVWXYZ012345';
   TRSP_LINE[24].LOT_NR_1 := 'ABCDEFGHIJKLMNOP';
   TRSP_LINE[24].LOT_NR_2 := 'ABCDEFGHIJKLMNOP';
   TRSP_LINE[24].LOT_NR_3 := 'ABCDEFGHIJKLMNOP';
   TRSP_LINE[25].ProductIdent := 'ABCDEFGHIJKLMNOP';
   TRSP_LINE[25].ProductName := 'ABCDEFGHIJKLMNOPQRSTUVWXYZ012345';
   TRSP_LINE[25].LOT_NR_1 := 'ABCDEFGHIJKLMNOP';
   TRSP_LINE[25].LOT_NR_2 := 'ABCDEFGHIJKLMNOP';
   TRSP_LINE[25].LOT_NR_3 := 'ABCDEFGHIJKLMNOP';
   TRSP_LINE[26].ProductIdent := 'ABCDEFGHIJKLMNOP';
   TRSP_LINE[26].ProductName := 'ABCDEFGHIJKLMNOPQRSTUVWXYZ012345';
   TRSP_LINE[26].LOT_NR_1 := 'ABCDEFGHIJKLMNOP';
   TRSP_LINE[26].LOT_NR_2 := 'ABCDEFGHIJKLMNOP';
   TRSP_LINE[26].LOT_NR_3 := 'ABCDEFGHIJKLMNOP';
   TRSP_LINE[27].ProductIdent := 'ABCDEFGHIJKLMNOP';
   TRSP_LINE[27].ProductName := 'ABCDEFGHIJKLMNOPQRSTUVWXYZ012345';
   TRSP_LINE[27].LOT_NR_1 := 'ABCDEFGHIJKLMNOP';
   TRSP_LINE[27].LOT_NR_2 := 'ABCDEFGHIJKLMNOP';
   TRSP_LINE[27].LOT_NR_3 := 'ABCDEFGHIJKLMNOP';
   TRSP_LINE[28].ProductIdent := 'ABCDEFGHIJKLMNOP';
   TRSP_LINE[28].ProductName := 'ABCDEFGHIJKLMNOPQRSTUVWXYZ012345';
   TRSP_LINE[28].LOT_NR_1 := 'ABCDEFGHIJKLMNOP';
   TRSP_LINE[28].LOT_NR_2 := 'ABCDEFGHIJKLMNOP';
   TRSP_LINE[28].LOT_NR_3 := 'ABCDEFGHIJKLMNOP';
   TRSP_LINE[29].ProductIdent := 'ABCDEFGHIJKLMNOP';
   TRSP_LINE[29].ProductName := 'ABCDEFGHIJKLMNOPQRSTUVWXYZ012345';
   TRSP_LINE[29].LOT_NR_1 := 'ABCDEFGHIJKLMNOP';
   TRSP_LINE[29].LOT_NR_2 := 'ABCDEFGHIJKLMNOP';
   TRSP_LINE[29].LOT_NR_3 := 'ABCDEFGHIJKLMNOP';
   TRSP_LINE[30].ProductIdent := 'ABCDEFGHIJKLMNOP';
   TRSP_LINE[30].ProductName := 'ABCDEFGHIJKLMNOPQRSTUVWXYZ012345';
   TRSP_LINE[30].LOT_NR_1 := 'ABCDEFGHIJKLMNOP';
   TRSP_LINE[30].LOT_NR_2 := 'ABCDEFGHIJKLMNOP';
   TRSP_LINE[30].LOT_NR_3 := 'ABCDEFGHIJKLMNOP';
   TRSP_LINE[31].ProductIdent := 'ABCDEFGHIJKLMNOP';
   TRSP_LINE[31].ProductName := 'ABCDEFGHIJKLMNOPQRSTUVWXYZ012345';
   TRSP_LINE[31].LOT_NR_1 := 'ABCDEFGHIJKLMNOP';
   TRSP_LINE[31].LOT_NR_2 := 'ABCDEFGHIJKLMNOP';
   TRSP_LINE[31].LOT_NR_3 := 'ABCDEFGHIJKLMNOP';
   TRSP_LINE[32].ProductIdent := 'ABCDEFGHIJKLMNOP';
   TRSP_LINE[32].ProductName := 'ABCDEFGHIJKLMNOPQRSTUVWXYZ012345';
   TRSP_LINE[32].LOT_NR_1 := 'ABCDEFGHIJKLMNOP';
   TRSP_LINE[32].LOT_NR_2 := 'ABCDEFGHIJKLMNOP';
   TRSP_LINE[32].LOT_NR_3 := 'ABCDEFGHIJKLMNOP';
END_DATA_BLOCK

DATA_BLOCK "ASW_HandAddInfoData"	// DB 83
TITLE = COPYRIGHT:    (C) 2003  BUHLER AG, CH-9240 UZWIL, SWITZERLAND
//
//PRODUCT:      GP_GCS7
//
//TITLE:        
//
//------------------------------------------------------------------------------------------------------
//
//IDENT:               AUTHOR:         DEPT:                 DATE:
//
//DB83.1A            CE                    FU53                    03.03.2003
//
//------------------------------------------------------------------------------------------------------
//
//PURPOSE:      MANUAL : see [MxxMAN]
//
//RESTRICTIONS: 
//------------------------------------------------------------------------------------------------------
//
//
//
//
//
AUTHOR : CE
FAMILY : USW
VERSION : 0.0
  STRUCT
   Reserve0 : ARRAY  [0 .. 99 ] OF BYTE ;
   HandAddition9xx : ARRAY  [1 .. 20 ] OF UDT 1004;
  END_STRUCT ;	
BEGIN
   HandAddition9xx[1].ProductIdent := 'ABCDEFGHIJKLMNOP';
   HandAddition9xx[1].ProductName := 'ABCDEFGHIJKLMNOPQRSTUVWXYZ012345';
   HandAddition9xx[1].Barcode := 'ABCDEFGHIJKLMNOPQRSTUVWXYZ012345';
   HandAddition9xx[2].ProductIdent := 'ABCDEFGHIJKLMNOP';
   HandAddition9xx[2].ProductName := 'ABCDEFGHIJKLMNOPQRSTUVWXYZ012345';
   HandAddition9xx[2].Barcode := 'ABCDEFGHIJKLMNOPQRSTUVWXYZ012345';
   HandAddition9xx[3].ProductIdent := 'ABCDEFGHIJKLMNOP';
   HandAddition9xx[3].ProductName := 'ABCDEFGHIJKLMNOPQRSTUVWXYZ012345';
   HandAddition9xx[3].Barcode := 'ABCDEFGHIJKLMNOPQRSTUVWXYZ012345';
   HandAddition9xx[4].ProductIdent := 'ABCDEFGHIJKLMNOP';
   HandAddition9xx[4].ProductName := 'ABCDEFGHIJKLMNOPQRSTUVWXYZ012345';
   HandAddition9xx[4].Barcode := 'ABCDEFGHIJKLMNOPQRSTUVWXYZ012345';
   HandAddition9xx[5].ProductIdent := 'ABCDEFGHIJKLMNOP';
   HandAddition9xx[5].ProductName := 'ABCDEFGHIJKLMNOPQRSTUVWXYZ012345';
   HandAddition9xx[5].Barcode := 'ABCDEFGHIJKLMNOPQRSTUVWXYZ012345';
   HandAddition9xx[6].ProductIdent := 'ABCDEFGHIJKLMNOP';
   HandAddition9xx[6].ProductName := 'ABCDEFGHIJKLMNOPQRSTUVWXYZ012345';
   HandAddition9xx[6].Barcode := 'ABCDEFGHIJKLMNOPQRSTUVWXYZ012345';
   HandAddition9xx[7].ProductIdent := 'ABCDEFGHIJKLMNOP';
   HandAddition9xx[7].ProductName := 'ABCDEFGHIJKLMNOPQRSTUVWXYZ012345';
   HandAddition9xx[7].Barcode := 'ABCDEFGHIJKLMNOPQRSTUVWXYZ012345';
   HandAddition9xx[8].ProductIdent := 'ABCDEFGHIJKLMNOP';
   HandAddition9xx[8].ProductName := 'ABCDEFGHIJKLMNOPQRSTUVWXYZ012345';
   HandAddition9xx[8].Barcode := 'ABCDEFGHIJKLMNOPQRSTUVWXYZ012345';
   HandAddition9xx[9].ProductIdent := 'ABCDEFGHIJKLMNOP';
   HandAddition9xx[9].ProductName := 'ABCDEFGHIJKLMNOPQRSTUVWXYZ012345';
   HandAddition9xx[9].Barcode := 'ABCDEFGHIJKLMNOPQRSTUVWXYZ012345';
   HandAddition9xx[10].ProductIdent := 'ABCDEFGHIJKLMNOP';
   HandAddition9xx[10].ProductName := 'ABCDEFGHIJKLMNOPQRSTUVWXYZ012345';
   HandAddition9xx[10].Barcode := 'ABCDEFGHIJKLMNOPQRSTUVWXYZ012345';
   HandAddition9xx[11].ProductIdent := 'ABCDEFGHIJKLMNOP';
   HandAddition9xx[11].ProductName := 'ABCDEFGHIJKLMNOPQRSTUVWXYZ012345';
   HandAddition9xx[11].Barcode := 'ABCDEFGHIJKLMNOPQRSTUVWXYZ012345';
   HandAddition9xx[12].ProductIdent := 'ABCDEFGHIJKLMNOP';
   HandAddition9xx[12].ProductName := 'ABCDEFGHIJKLMNOPQRSTUVWXYZ012345';
   HandAddition9xx[12].Barcode := 'ABCDEFGHIJKLMNOPQRSTUVWXYZ012345';
   HandAddition9xx[13].ProductIdent := 'ABCDEFGHIJKLMNOP';
   HandAddition9xx[13].ProductName := 'ABCDEFGHIJKLMNOPQRSTUVWXYZ012345';
   HandAddition9xx[13].Barcode := 'ABCDEFGHIJKLMNOPQRSTUVWXYZ012345';
   HandAddition9xx[14].ProductIdent := 'ABCDEFGHIJKLMNOP';
   HandAddition9xx[14].ProductName := 'ABCDEFGHIJKLMNOPQRSTUVWXYZ012345';
   HandAddition9xx[14].Barcode := 'ABCDEFGHIJKLMNOPQRSTUVWXYZ012345';
   HandAddition9xx[15].ProductIdent := 'ABCDEFGHIJKLMNOP';
   HandAddition9xx[15].ProductName := 'ABCDEFGHIJKLMNOPQRSTUVWXYZ012345';
   HandAddition9xx[15].Barcode := 'ABCDEFGHIJKLMNOPQRSTUVWXYZ012345';
   HandAddition9xx[16].ProductIdent := 'ABCDEFGHIJKLMNOP';
   HandAddition9xx[16].ProductName := 'ABCDEFGHIJKLMNOPQRSTUVWXYZ012345';
   HandAddition9xx[16].Barcode := 'ABCDEFGHIJKLMNOPQRSTUVWXYZ012345';
   HandAddition9xx[17].ProductIdent := 'ABCDEFGHIJKLMNOP';
   HandAddition9xx[17].ProductName := 'ABCDEFGHIJKLMNOPQRSTUVWXYZ012345';
   HandAddition9xx[17].Barcode := 'ABCDEFGHIJKLMNOPQRSTUVWXYZ012345';
   HandAddition9xx[18].ProductIdent := 'ABCDEFGHIJKLMNOP';
   HandAddition9xx[18].ProductName := 'ABCDEFGHIJKLMNOPQRSTUVWXYZ012345';
   HandAddition9xx[18].Barcode := 'ABCDEFGHIJKLMNOPQRSTUVWXYZ012345';
   HandAddition9xx[19].ProductIdent := 'ABCDEFGHIJKLMNOP';
   HandAddition9xx[19].ProductName := 'ABCDEFGHIJKLMNOPQRSTUVWXYZ012345';
   HandAddition9xx[19].Barcode := 'ABCDEFGHIJKLMNOPQRSTUVWXYZ012345';
   HandAddition9xx[20].ProductIdent := 'ABCDEFGHIJKLMNOP';
   HandAddition9xx[20].ProductName := 'ABCDEFGHIJKLMNOPQRSTUVWXYZ012345';
   HandAddition9xx[20].Barcode := 'ABCDEFGHIJKLMNOPQRSTUVWXYZ012345';
END_DATA_BLOCK

DATA_BLOCK "PCC_YieldScaleDB"	// DB 90
TITLE = COPYRIGHT:    (C) 2000 BY  BUHLER AG
//                           CH-9240 UZWIL  SWITZERLAND
//
//PRODUCT:      MELE_ZZZ01_xx
//
//TITLE:        Scale data for the PCC yield calculator
//
//              Waagendaten für den PCC-Ausbeuterechner
//
//
//--------------------------------------------------------------------------------
//
//IDENT:         AUTHOR:             DEPT:                             DATE:
//
//P01_DB1013.1.0 Ph. Engler          MU664                             04-Okt-2000
//               1st Release
//
//--------------------------------------------------------------------------------
//
//PURPOSE:      
//
//RESTRICTIONS: 
//
//--------------------------------------------------------------------------------
//
//
AUTHOR : PE
FAMILY : USW
VERSION : 1.0
  STRUCT
   PCWrite : STRUCT
    Hsk : STRUCT
     Q_Status : BOOL ;
    END_STRUCT ;
   END_STRUCT ;
   PCRead : STRUCT
    Hsk : STRUCT
     F_Status : BOOL ;
    END_STRUCT ;
    _x_xx1WE : UDT 19000;	//Use this UDT for MELE Hostsystems
    _x_xx2WE : UDT 19001;	//Use this UDT for WinCoS Hostsystems
   END_STRUCT ;
  END_STRUCT ;	
BEGIN
END_DATA_BLOCK

DATA_BLOCK "ASW_DFCATargData"	// DB 480
TITLE = COPYRIGHT:    (C) 2003  BUHLER AG, CH-9240 UZWIL, SWITZERLAND
//
//PRODUCT:      GP_GCS7
//
//TITLE:        
//
//------------------------------------------------------------------------------------------------------
//
//IDENT:               AUTHOR:         DEPT:                 DATE:
//
//DB720.1A           CE                    FU53                    03.03.2003
//
//------------------------------------------------------------------------------------------------------
//
//PURPOSE:      MANUAL : see [MxxMAN]
//
//RESTRICTIONS: 
//------------------------------------------------------------------------------------------------------
//
//
AUTHOR : CE
FAMILY : USW
VERSION : 0.0
  STRUCT
   Reserve0 : ARRAY  [0 .. 99 ] OF BYTE ;
   Line : ARRAY  [11 .. 32 ] OF UDT 1005;
  END_STRUCT ;	
BEGIN
   Line[11].DFCx.PelletingDieName[1] := ' ';
   Line[11].DFCx.PelletingDieName[2] := ' ';
   Line[11].DFCx.PelletingDieName[3] := ' ';
   Line[11].DFCx.PelletingDieName[4] := ' ';
   Line[11].DFCx.PelletingDieName[5] := ' ';
   Line[11].DFCx.PelletingDieName[6] := ' ';
   Line[11].DFCx.PelletingDieName[7] := ' ';
   Line[11].DFCx.PelletingDieName[8] := ' ';
   Line[11].DFCx.PelletingDieName[9] := ' ';
   Line[11].DFCx.PelletingDieName[10] := ' ';
   Line[11].DFCx.ParameterSetIdent[1] := ' ';
   Line[11].DFCx.ParameterSetIdent[2] := ' ';
   Line[11].DFCx.ParameterSetIdent[3] := ' ';
   Line[11].DFCx.ParameterSetIdent[4] := ' ';
   Line[11].DFCx.ParameterSetIdent[5] := ' ';
   Line[11].DFCx.ParameterSetIdent[6] := ' ';
   Line[11].DFCx.ParameterSetIdent[7] := ' ';
   Line[11].DFCx.ParameterSetIdent[8] := ' ';
   Line[11].DFCx.ParameterSetIdent[9] := ' ';
   Line[11].DFCx.ParameterSetIdent[10] := ' ';
   Line[11].DFCx.ParameterSetIdent[11] := ' ';
   Line[11].DFCx.ParameterSetIdent[12] := ' ';
   Line[11].DFCx.ParameterSetIdent[13] := ' ';
   Line[11].DFCx.ParameterSetIdent[14] := ' ';
   Line[11].DFCx.ParameterSetIdent[15] := ' ';
   Line[11].DFCx.ParameterSetIdent[16] := ' ';
   Line[11].DFCx.ParameterSetName[1] := ' ';
   Line[11].DFCx.ParameterSetName[2] := ' ';
   Line[11].DFCx.ParameterSetName[3] := ' ';
   Line[11].DFCx.ParameterSetName[4] := ' ';
   Line[11].DFCx.ParameterSetName[5] := ' ';
   Line[11].DFCx.ParameterSetName[6] := ' ';
   Line[11].DFCx.ParameterSetName[7] := ' ';
   Line[11].DFCx.ParameterSetName[8] := ' ';
   Line[11].DFCx.ParameterSetName[9] := ' ';
   Line[11].DFCx.ParameterSetName[10] := ' ';
   Line[11].DFCx.ParameterSetName[11] := ' ';
   Line[11].DFCx.ParameterSetName[12] := ' ';
   Line[11].DFCx.ParameterSetName[13] := ' ';
   Line[11].DFCx.ParameterSetName[14] := ' ';
   Line[11].DFCx.ParameterSetName[15] := ' ';
   Line[11].DFCx.ParameterSetName[16] := ' ';
   Line[11].DFCx.ParameterSetName[17] := ' ';
   Line[11].DFCx.ParameterSetName[18] := ' ';
   Line[11].DFCx.ParameterSetName[19] := ' ';
   Line[11].DFCx.ParameterSetName[20] := ' ';
   Line[11].DFCx.ParameterSetName[21] := ' ';
   Line[11].DFCx.ParameterSetName[22] := ' ';
   Line[11].DFCx.ParameterSetName[23] := ' ';
   Line[11].DFCx.ParameterSetName[24] := ' ';
   Line[11].DFCx.ParameterSetName[25] := ' ';
   Line[11].DFCx.ParameterSetName[26] := ' ';
   Line[11].DFCx.ParameterSetName[27] := ' ';
   Line[11].DFCx.ParameterSetName[28] := ' ';
   Line[11].DFCx.ParameterSetName[29] := ' ';
   Line[11].DFCx.ParameterSetName[30] := ' ';
   Line[12].DFCx.PelletingDieName[1] := ' ';
   Line[12].DFCx.PelletingDieName[2] := ' ';
   Line[12].DFCx.PelletingDieName[3] := ' ';
   Line[12].DFCx.PelletingDieName[4] := ' ';
   Line[12].DFCx.PelletingDieName[5] := ' ';
   Line[12].DFCx.PelletingDieName[6] := ' ';
   Line[12].DFCx.PelletingDieName[7] := ' ';
   Line[12].DFCx.PelletingDieName[8] := ' ';
   Line[12].DFCx.PelletingDieName[9] := ' ';
   Line[12].DFCx.PelletingDieName[10] := ' ';
   Line[12].DFCx.ParameterSetIdent[1] := ' ';
   Line[12].DFCx.ParameterSetIdent[2] := ' ';
   Line[12].DFCx.ParameterSetIdent[3] := ' ';
   Line[12].DFCx.ParameterSetIdent[4] := ' ';
   Line[12].DFCx.ParameterSetIdent[5] := ' ';
   Line[12].DFCx.ParameterSetIdent[6] := ' ';
   Line[12].DFCx.ParameterSetIdent[7] := ' ';
   Line[12].DFCx.ParameterSetIdent[8] := ' ';
   Line[12].DFCx.ParameterSetIdent[9] := ' ';
   Line[12].DFCx.ParameterSetIdent[10] := ' ';
   Line[12].DFCx.ParameterSetIdent[11] := ' ';
   Line[12].DFCx.ParameterSetIdent[12] := ' ';
   Line[12].DFCx.ParameterSetIdent[13] := ' ';
   Line[12].DFCx.ParameterSetIdent[14] := ' ';
   Line[12].DFCx.ParameterSetIdent[15] := ' ';
   Line[12].DFCx.ParameterSetIdent[16] := ' ';
   Line[12].DFCx.ParameterSetName[1] := ' ';
   Line[12].DFCx.ParameterSetName[2] := ' ';
   Line[12].DFCx.ParameterSetName[3] := ' ';
   Line[12].DFCx.ParameterSetName[4] := ' ';
   Line[12].DFCx.ParameterSetName[5] := ' ';
   Line[12].DFCx.ParameterSetName[6] := ' ';
   Line[12].DFCx.ParameterSetName[7] := ' ';
   Line[12].DFCx.ParameterSetName[8] := ' ';
   Line[12].DFCx.ParameterSetName[9] := ' ';
   Line[12].DFCx.ParameterSetName[10] := ' ';
   Line[12].DFCx.ParameterSetName[11] := ' ';
   Line[12].DFCx.ParameterSetName[12] := ' ';
   Line[12].DFCx.ParameterSetName[13] := ' ';
   Line[12].DFCx.ParameterSetName[14] := ' ';
   Line[12].DFCx.ParameterSetName[15] := ' ';
   Line[12].DFCx.ParameterSetName[16] := ' ';
   Line[12].DFCx.ParameterSetName[17] := ' ';
   Line[12].DFCx.ParameterSetName[18] := ' ';
   Line[12].DFCx.ParameterSetName[19] := ' ';
   Line[12].DFCx.ParameterSetName[20] := ' ';
   Line[12].DFCx.ParameterSetName[21] := ' ';
   Line[12].DFCx.ParameterSetName[22] := ' ';
   Line[12].DFCx.ParameterSetName[23] := ' ';
   Line[12].DFCx.ParameterSetName[24] := ' ';
   Line[12].DFCx.ParameterSetName[25] := ' ';
   Line[12].DFCx.ParameterSetName[26] := ' ';
   Line[12].DFCx.ParameterSetName[27] := ' ';
   Line[12].DFCx.ParameterSetName[28] := ' ';
   Line[12].DFCx.ParameterSetName[29] := ' ';
   Line[12].DFCx.ParameterSetName[30] := ' ';
   Line[13].DFCx.PelletingDieName[1] := ' ';
   Line[13].DFCx.PelletingDieName[2] := ' ';
   Line[13].DFCx.PelletingDieName[3] := ' ';
   Line[13].DFCx.PelletingDieName[4] := ' ';
   Line[13].DFCx.PelletingDieName[5] := ' ';
   Line[13].DFCx.PelletingDieName[6] := ' ';
   Line[13].DFCx.PelletingDieName[7] := ' ';
   Line[13].DFCx.PelletingDieName[8] := ' ';
   Line[13].DFCx.PelletingDieName[9] := ' ';
   Line[13].DFCx.PelletingDieName[10] := ' ';
   Line[13].DFCx.ParameterSetIdent[1] := ' ';
   Line[13].DFCx.ParameterSetIdent[2] := ' ';
   Line[13].DFCx.ParameterSetIdent[3] := ' ';
   Line[13].DFCx.ParameterSetIdent[4] := ' ';
   Line[13].DFCx.ParameterSetIdent[5] := ' ';
   Line[13].DFCx.ParameterSetIdent[6] := ' ';
   Line[13].DFCx.ParameterSetIdent[7] := ' ';
   Line[13].DFCx.ParameterSetIdent[8] := ' ';
   Line[13].DFCx.ParameterSetIdent[9] := ' ';
   Line[13].DFCx.ParameterSetIdent[10] := ' ';
   Line[13].DFCx.ParameterSetIdent[11] := ' ';
   Line[13].DFCx.ParameterSetIdent[12] := ' ';
   Line[13].DFCx.ParameterSetIdent[13] := ' ';
   Line[13].DFCx.ParameterSetIdent[14] := ' ';
   Line[13].DFCx.ParameterSetIdent[15] := ' ';
   Line[13].DFCx.ParameterSetIdent[16] := ' ';
   Line[13].DFCx.ParameterSetName[1] := ' ';
   Line[13].DFCx.ParameterSetName[2] := ' ';
   Line[13].DFCx.ParameterSetName[3] := ' ';
   Line[13].DFCx.ParameterSetName[4] := ' ';
   Line[13].DFCx.ParameterSetName[5] := ' ';
   Line[13].DFCx.ParameterSetName[6] := ' ';
   Line[13].DFCx.ParameterSetName[7] := ' ';
   Line[13].DFCx.ParameterSetName[8] := ' ';
   Line[13].DFCx.ParameterSetName[9] := ' ';
   Line[13].DFCx.ParameterSetName[10] := ' ';
   Line[13].DFCx.ParameterSetName[11] := ' ';
   Line[13].DFCx.ParameterSetName[12] := ' ';
   Line[13].DFCx.ParameterSetName[13] := ' ';
   Line[13].DFCx.ParameterSetName[14] := ' ';
   Line[13].DFCx.ParameterSetName[15] := ' ';
   Line[13].DFCx.ParameterSetName[16] := ' ';
   Line[13].DFCx.ParameterSetName[17] := ' ';
   Line[13].DFCx.ParameterSetName[18] := ' ';
   Line[13].DFCx.ParameterSetName[19] := ' ';
   Line[13].DFCx.ParameterSetName[20] := ' ';
   Line[13].DFCx.ParameterSetName[21] := ' ';
   Line[13].DFCx.ParameterSetName[22] := ' ';
   Line[13].DFCx.ParameterSetName[23] := ' ';
   Line[13].DFCx.ParameterSetName[24] := ' ';
   Line[13].DFCx.ParameterSetName[25] := ' ';
   Line[13].DFCx.ParameterSetName[26] := ' ';
   Line[13].DFCx.ParameterSetName[27] := ' ';
   Line[13].DFCx.ParameterSetName[28] := ' ';
   Line[13].DFCx.ParameterSetName[29] := ' ';
   Line[13].DFCx.ParameterSetName[30] := ' ';
   Line[14].DFCx.PelletingDieName[1] := ' ';
   Line[14].DFCx.PelletingDieName[2] := ' ';
   Line[14].DFCx.PelletingDieName[3] := ' ';
   Line[14].DFCx.PelletingDieName[4] := ' ';
   Line[14].DFCx.PelletingDieName[5] := ' ';
   Line[14].DFCx.PelletingDieName[6] := ' ';
   Line[14].DFCx.PelletingDieName[7] := ' ';
   Line[14].DFCx.PelletingDieName[8] := ' ';
   Line[14].DFCx.PelletingDieName[9] := ' ';
   Line[14].DFCx.PelletingDieName[10] := ' ';
   Line[14].DFCx.ParameterSetIdent[1] := ' ';
   Line[14].DFCx.ParameterSetIdent[2] := ' ';
   Line[14].DFCx.ParameterSetIdent[3] := ' ';
   Line[14].DFCx.ParameterSetIdent[4] := ' ';
   Line[14].DFCx.ParameterSetIdent[5] := ' ';
   Line[14].DFCx.ParameterSetIdent[6] := ' ';
   Line[14].DFCx.ParameterSetIdent[7] := ' ';
   Line[14].DFCx.ParameterSetIdent[8] := ' ';
   Line[14].DFCx.ParameterSetIdent[9] := ' ';
   Line[14].DFCx.ParameterSetIdent[10] := ' ';
   Line[14].DFCx.ParameterSetIdent[11] := ' ';
   Line[14].DFCx.ParameterSetIdent[12] := ' ';
   Line[14].DFCx.ParameterSetIdent[13] := ' ';
   Line[14].DFCx.ParameterSetIdent[14] := ' ';
   Line[14].DFCx.ParameterSetIdent[15] := ' ';
   Line[14].DFCx.ParameterSetIdent[16] := ' ';
   Line[14].DFCx.ParameterSetName[1] := ' ';
   Line[14].DFCx.ParameterSetName[2] := ' ';
   Line[14].DFCx.ParameterSetName[3] := ' ';
   Line[14].DFCx.ParameterSetName[4] := ' ';
   Line[14].DFCx.ParameterSetName[5] := ' ';
   Line[14].DFCx.ParameterSetName[6] := ' ';
   Line[14].DFCx.ParameterSetName[7] := ' ';
   Line[14].DFCx.ParameterSetName[8] := ' ';
   Line[14].DFCx.ParameterSetName[9] := ' ';
   Line[14].DFCx.ParameterSetName[10] := ' ';
   Line[14].DFCx.ParameterSetName[11] := ' ';
   Line[14].DFCx.ParameterSetName[12] := ' ';
   Line[14].DFCx.ParameterSetName[13] := ' ';
   Line[14].DFCx.ParameterSetName[14] := ' ';
   Line[14].DFCx.ParameterSetName[15] := ' ';
   Line[14].DFCx.ParameterSetName[16] := ' ';
   Line[14].DFCx.ParameterSetName[17] := ' ';
   Line[14].DFCx.ParameterSetName[18] := ' ';
   Line[14].DFCx.ParameterSetName[19] := ' ';
   Line[14].DFCx.ParameterSetName[20] := ' ';
   Line[14].DFCx.ParameterSetName[21] := ' ';
   Line[14].DFCx.ParameterSetName[22] := ' ';
   Line[14].DFCx.ParameterSetName[23] := ' ';
   Line[14].DFCx.ParameterSetName[24] := ' ';
   Line[14].DFCx.ParameterSetName[25] := ' ';
   Line[14].DFCx.ParameterSetName[26] := ' ';
   Line[14].DFCx.ParameterSetName[27] := ' ';
   Line[14].DFCx.ParameterSetName[28] := ' ';
   Line[14].DFCx.ParameterSetName[29] := ' ';
   Line[14].DFCx.ParameterSetName[30] := ' ';
   Line[15].DFCx.PelletingDieName[1] := ' ';
   Line[15].DFCx.PelletingDieName[2] := ' ';
   Line[15].DFCx.PelletingDieName[3] := ' ';
   Line[15].DFCx.PelletingDieName[4] := ' ';
   Line[15].DFCx.PelletingDieName[5] := ' ';
   Line[15].DFCx.PelletingDieName[6] := ' ';
   Line[15].DFCx.PelletingDieName[7] := ' ';
   Line[15].DFCx.PelletingDieName[8] := ' ';
   Line[15].DFCx.PelletingDieName[9] := ' ';
   Line[15].DFCx.PelletingDieName[10] := ' ';
   Line[15].DFCx.ParameterSetIdent[1] := ' ';
   Line[15].DFCx.ParameterSetIdent[2] := ' ';
   Line[15].DFCx.ParameterSetIdent[3] := ' ';
   Line[15].DFCx.ParameterSetIdent[4] := ' ';
   Line[15].DFCx.ParameterSetIdent[5] := ' ';
   Line[15].DFCx.ParameterSetIdent[6] := ' ';
   Line[15].DFCx.ParameterSetIdent[7] := ' ';
   Line[15].DFCx.ParameterSetIdent[8] := ' ';
   Line[15].DFCx.ParameterSetIdent[9] := ' ';
   Line[15].DFCx.ParameterSetIdent[10] := ' ';
   Line[15].DFCx.ParameterSetIdent[11] := ' ';
   Line[15].DFCx.ParameterSetIdent[12] := ' ';
   Line[15].DFCx.ParameterSetIdent[13] := ' ';
   Line[15].DFCx.ParameterSetIdent[14] := ' ';
   Line[15].DFCx.ParameterSetIdent[15] := ' ';
   Line[15].DFCx.ParameterSetIdent[16] := ' ';
   Line[15].DFCx.ParameterSetName[1] := ' ';
   Line[15].DFCx.ParameterSetName[2] := ' ';
   Line[15].DFCx.ParameterSetName[3] := ' ';
   Line[15].DFCx.ParameterSetName[4] := ' ';
   Line[15].DFCx.ParameterSetName[5] := ' ';
   Line[15].DFCx.ParameterSetName[6] := ' ';
   Line[15].DFCx.ParameterSetName[7] := ' ';
   Line[15].DFCx.ParameterSetName[8] := ' ';
   Line[15].DFCx.ParameterSetName[9] := ' ';
   Line[15].DFCx.ParameterSetName[10] := ' ';
   Line[15].DFCx.ParameterSetName[11] := ' ';
   Line[15].DFCx.ParameterSetName[12] := ' ';
   Line[15].DFCx.ParameterSetName[13] := ' ';
   Line[15].DFCx.ParameterSetName[14] := ' ';
   Line[15].DFCx.ParameterSetName[15] := ' ';
   Line[15].DFCx.ParameterSetName[16] := ' ';
   Line[15].DFCx.ParameterSetName[17] := ' ';
   Line[15].DFCx.ParameterSetName[18] := ' ';
   Line[15].DFCx.ParameterSetName[19] := ' ';
   Line[15].DFCx.ParameterSetName[20] := ' ';
   Line[15].DFCx.ParameterSetName[21] := ' ';
   Line[15].DFCx.ParameterSetName[22] := ' ';
   Line[15].DFCx.ParameterSetName[23] := ' ';
   Line[15].DFCx.ParameterSetName[24] := ' ';
   Line[15].DFCx.ParameterSetName[25] := ' ';
   Line[15].DFCx.ParameterSetName[26] := ' ';
   Line[15].DFCx.ParameterSetName[27] := ' ';
   Line[15].DFCx.ParameterSetName[28] := ' ';
   Line[15].DFCx.ParameterSetName[29] := ' ';
   Line[15].DFCx.ParameterSetName[30] := ' ';
   Line[16].DFCx.PelletingDieName[1] := ' ';
   Line[16].DFCx.PelletingDieName[2] := ' ';
   Line[16].DFCx.PelletingDieName[3] := ' ';
   Line[16].DFCx.PelletingDieName[4] := ' ';
   Line[16].DFCx.PelletingDieName[5] := ' ';
   Line[16].DFCx.PelletingDieName[6] := ' ';
   Line[16].DFCx.PelletingDieName[7] := ' ';
   Line[16].DFCx.PelletingDieName[8] := ' ';
   Line[16].DFCx.PelletingDieName[9] := ' ';
   Line[16].DFCx.PelletingDieName[10] := ' ';
   Line[16].DFCx.ParameterSetIdent[1] := ' ';
   Line[16].DFCx.ParameterSetIdent[2] := ' ';
   Line[16].DFCx.ParameterSetIdent[3] := ' ';
   Line[16].DFCx.ParameterSetIdent[4] := ' ';
   Line[16].DFCx.ParameterSetIdent[5] := ' ';
   Line[16].DFCx.ParameterSetIdent[6] := ' ';
   Line[16].DFCx.ParameterSetIdent[7] := ' ';
   Line[16].DFCx.ParameterSetIdent[8] := ' ';
   Line[16].DFCx.ParameterSetIdent[9] := ' ';
   Line[16].DFCx.ParameterSetIdent[10] := ' ';
   Line[16].DFCx.ParameterSetIdent[11] := ' ';
   Line[16].DFCx.ParameterSetIdent[12] := ' ';
   Line[16].DFCx.ParameterSetIdent[13] := ' ';
   Line[16].DFCx.ParameterSetIdent[14] := ' ';
   Line[16].DFCx.ParameterSetIdent[15] := ' ';
   Line[16].DFCx.ParameterSetIdent[16] := ' ';
   Line[16].DFCx.ParameterSetName[1] := ' ';
   Line[16].DFCx.ParameterSetName[2] := ' ';
   Line[16].DFCx.ParameterSetName[3] := ' ';
   Line[16].DFCx.ParameterSetName[4] := ' ';
   Line[16].DFCx.ParameterSetName[5] := ' ';
   Line[16].DFCx.ParameterSetName[6] := ' ';
   Line[16].DFCx.ParameterSetName[7] := ' ';
   Line[16].DFCx.ParameterSetName[8] := ' ';
   Line[16].DFCx.ParameterSetName[9] := ' ';
   Line[16].DFCx.ParameterSetName[10] := ' ';
   Line[16].DFCx.ParameterSetName[11] := ' ';
   Line[16].DFCx.ParameterSetName[12] := ' ';
   Line[16].DFCx.ParameterSetName[13] := ' ';
   Line[16].DFCx.ParameterSetName[14] := ' ';
   Line[16].DFCx.ParameterSetName[15] := ' ';
   Line[16].DFCx.ParameterSetName[16] := ' ';
   Line[16].DFCx.ParameterSetName[17] := ' ';
   Line[16].DFCx.ParameterSetName[18] := ' ';
   Line[16].DFCx.ParameterSetName[19] := ' ';
   Line[16].DFCx.ParameterSetName[20] := ' ';
   Line[16].DFCx.ParameterSetName[21] := ' ';
   Line[16].DFCx.ParameterSetName[22] := ' ';
   Line[16].DFCx.ParameterSetName[23] := ' ';
   Line[16].DFCx.ParameterSetName[24] := ' ';
   Line[16].DFCx.ParameterSetName[25] := ' ';
   Line[16].DFCx.ParameterSetName[26] := ' ';
   Line[16].DFCx.ParameterSetName[27] := ' ';
   Line[16].DFCx.ParameterSetName[28] := ' ';
   Line[16].DFCx.ParameterSetName[29] := ' ';
   Line[16].DFCx.ParameterSetName[30] := ' ';
   Line[17].DFCx.PelletingDieName[1] := ' ';
   Line[17].DFCx.PelletingDieName[2] := ' ';
   Line[17].DFCx.PelletingDieName[3] := ' ';
   Line[17].DFCx.PelletingDieName[4] := ' ';
   Line[17].DFCx.PelletingDieName[5] := ' ';
   Line[17].DFCx.PelletingDieName[6] := ' ';
   Line[17].DFCx.PelletingDieName[7] := ' ';
   Line[17].DFCx.PelletingDieName[8] := ' ';
   Line[17].DFCx.PelletingDieName[9] := ' ';
   Line[17].DFCx.PelletingDieName[10] := ' ';
   Line[17].DFCx.ParameterSetIdent[1] := ' ';
   Line[17].DFCx.ParameterSetIdent[2] := ' ';
   Line[17].DFCx.ParameterSetIdent[3] := ' ';
   Line[17].DFCx.ParameterSetIdent[4] := ' ';
   Line[17].DFCx.ParameterSetIdent[5] := ' ';
   Line[17].DFCx.ParameterSetIdent[6] := ' ';
   Line[17].DFCx.ParameterSetIdent[7] := ' ';
   Line[17].DFCx.ParameterSetIdent[8] := ' ';
   Line[17].DFCx.ParameterSetIdent[9] := ' ';
   Line[17].DFCx.ParameterSetIdent[10] := ' ';
   Line[17].DFCx.ParameterSetIdent[11] := ' ';
   Line[17].DFCx.ParameterSetIdent[12] := ' ';
   Line[17].DFCx.ParameterSetIdent[13] := ' ';
   Line[17].DFCx.ParameterSetIdent[14] := ' ';
   Line[17].DFCx.ParameterSetIdent[15] := ' ';
   Line[17].DFCx.ParameterSetIdent[16] := ' ';
   Line[17].DFCx.ParameterSetName[1] := ' ';
   Line[17].DFCx.ParameterSetName[2] := ' ';
   Line[17].DFCx.ParameterSetName[3] := ' ';
   Line[17].DFCx.ParameterSetName[4] := ' ';
   Line[17].DFCx.ParameterSetName[5] := ' ';
   Line[17].DFCx.ParameterSetName[6] := ' ';
   Line[17].DFCx.ParameterSetName[7] := ' ';
   Line[17].DFCx.ParameterSetName[8] := ' ';
   Line[17].DFCx.ParameterSetName[9] := ' ';
   Line[17].DFCx.ParameterSetName[10] := ' ';
   Line[17].DFCx.ParameterSetName[11] := ' ';
   Line[17].DFCx.ParameterSetName[12] := ' ';
   Line[17].DFCx.ParameterSetName[13] := ' ';
   Line[17].DFCx.ParameterSetName[14] := ' ';
   Line[17].DFCx.ParameterSetName[15] := ' ';
   Line[17].DFCx.ParameterSetName[16] := ' ';
   Line[17].DFCx.ParameterSetName[17] := ' ';
   Line[17].DFCx.ParameterSetName[18] := ' ';
   Line[17].DFCx.ParameterSetName[19] := ' ';
   Line[17].DFCx.ParameterSetName[20] := ' ';
   Line[17].DFCx.ParameterSetName[21] := ' ';
   Line[17].DFCx.ParameterSetName[22] := ' ';
   Line[17].DFCx.ParameterSetName[23] := ' ';
   Line[17].DFCx.ParameterSetName[24] := ' ';
   Line[17].DFCx.ParameterSetName[25] := ' ';
   Line[17].DFCx.ParameterSetName[26] := ' ';
   Line[17].DFCx.ParameterSetName[27] := ' ';
   Line[17].DFCx.ParameterSetName[28] := ' ';
   Line[17].DFCx.ParameterSetName[29] := ' ';
   Line[17].DFCx.ParameterSetName[30] := ' ';
   Line[18].DFCx.PelletingDieName[1] := ' ';
   Line[18].DFCx.PelletingDieName[2] := ' ';
   Line[18].DFCx.PelletingDieName[3] := ' ';
   Line[18].DFCx.PelletingDieName[4] := ' ';
   Line[18].DFCx.PelletingDieName[5] := ' ';
   Line[18].DFCx.PelletingDieName[6] := ' ';
   Line[18].DFCx.PelletingDieName[7] := ' ';
   Line[18].DFCx.PelletingDieName[8] := ' ';
   Line[18].DFCx.PelletingDieName[9] := ' ';
   Line[18].DFCx.PelletingDieName[10] := ' ';
   Line[18].DFCx.ParameterSetIdent[1] := ' ';
   Line[18].DFCx.ParameterSetIdent[2] := ' ';
   Line[18].DFCx.ParameterSetIdent[3] := ' ';
   Line[18].DFCx.ParameterSetIdent[4] := ' ';
   Line[18].DFCx.ParameterSetIdent[5] := ' ';
   Line[18].DFCx.ParameterSetIdent[6] := ' ';
   Line[18].DFCx.ParameterSetIdent[7] := ' ';
   Line[18].DFCx.ParameterSetIdent[8] := ' ';
   Line[18].DFCx.ParameterSetIdent[9] := ' ';
   Line[18].DFCx.ParameterSetIdent[10] := ' ';
   Line[18].DFCx.ParameterSetIdent[11] := ' ';
   Line[18].DFCx.ParameterSetIdent[12] := ' ';
   Line[18].DFCx.ParameterSetIdent[13] := ' ';
   Line[18].DFCx.ParameterSetIdent[14] := ' ';
   Line[18].DFCx.ParameterSetIdent[15] := ' ';
   Line[18].DFCx.ParameterSetIdent[16] := ' ';
   Line[18].DFCx.ParameterSetName[1] := ' ';
   Line[18].DFCx.ParameterSetName[2] := ' ';
   Line[18].DFCx.ParameterSetName[3] := ' ';
   Line[18].DFCx.ParameterSetName[4] := ' ';
   Line[18].DFCx.ParameterSetName[5] := ' ';
   Line[18].DFCx.ParameterSetName[6] := ' ';
   Line[18].DFCx.ParameterSetName[7] := ' ';
   Line[18].DFCx.ParameterSetName[8] := ' ';
   Line[18].DFCx.ParameterSetName[9] := ' ';
   Line[18].DFCx.ParameterSetName[10] := ' ';
   Line[18].DFCx.ParameterSetName[11] := ' ';
   Line[18].DFCx.ParameterSetName[12] := ' ';
   Line[18].DFCx.ParameterSetName[13] := ' ';
   Line[18].DFCx.ParameterSetName[14] := ' ';
   Line[18].DFCx.ParameterSetName[15] := ' ';
   Line[18].DFCx.ParameterSetName[16] := ' ';
   Line[18].DFCx.ParameterSetName[17] := ' ';
   Line[18].DFCx.ParameterSetName[18] := ' ';
   Line[18].DFCx.ParameterSetName[19] := ' ';
   Line[18].DFCx.ParameterSetName[20] := ' ';
   Line[18].DFCx.ParameterSetName[21] := ' ';
   Line[18].DFCx.ParameterSetName[22] := ' ';
   Line[18].DFCx.ParameterSetName[23] := ' ';
   Line[18].DFCx.ParameterSetName[24] := ' ';
   Line[18].DFCx.ParameterSetName[25] := ' ';
   Line[18].DFCx.ParameterSetName[26] := ' ';
   Line[18].DFCx.ParameterSetName[27] := ' ';
   Line[18].DFCx.ParameterSetName[28] := ' ';
   Line[18].DFCx.ParameterSetName[29] := ' ';
   Line[18].DFCx.ParameterSetName[30] := ' ';
   Line[19].DFCx.PelletingDieName[1] := ' ';
   Line[19].DFCx.PelletingDieName[2] := ' ';
   Line[19].DFCx.PelletingDieName[3] := ' ';
   Line[19].DFCx.PelletingDieName[4] := ' ';
   Line[19].DFCx.PelletingDieName[5] := ' ';
   Line[19].DFCx.PelletingDieName[6] := ' ';
   Line[19].DFCx.PelletingDieName[7] := ' ';
   Line[19].DFCx.PelletingDieName[8] := ' ';
   Line[19].DFCx.PelletingDieName[9] := ' ';
   Line[19].DFCx.PelletingDieName[10] := ' ';
   Line[19].DFCx.ParameterSetIdent[1] := ' ';
   Line[19].DFCx.ParameterSetIdent[2] := ' ';
   Line[19].DFCx.ParameterSetIdent[3] := ' ';
   Line[19].DFCx.ParameterSetIdent[4] := ' ';
   Line[19].DFCx.ParameterSetIdent[5] := ' ';
   Line[19].DFCx.ParameterSetIdent[6] := ' ';
   Line[19].DFCx.ParameterSetIdent[7] := ' ';
   Line[19].DFCx.ParameterSetIdent[8] := ' ';
   Line[19].DFCx.ParameterSetIdent[9] := ' ';
   Line[19].DFCx.ParameterSetIdent[10] := ' ';
   Line[19].DFCx.ParameterSetIdent[11] := ' ';
   Line[19].DFCx.ParameterSetIdent[12] := ' ';
   Line[19].DFCx.ParameterSetIdent[13] := ' ';
   Line[19].DFCx.ParameterSetIdent[14] := ' ';
   Line[19].DFCx.ParameterSetIdent[15] := ' ';
   Line[19].DFCx.ParameterSetIdent[16] := ' ';
   Line[19].DFCx.ParameterSetName[1] := ' ';
   Line[19].DFCx.ParameterSetName[2] := ' ';
   Line[19].DFCx.ParameterSetName[3] := ' ';
   Line[19].DFCx.ParameterSetName[4] := ' ';
   Line[19].DFCx.ParameterSetName[5] := ' ';
   Line[19].DFCx.ParameterSetName[6] := ' ';
   Line[19].DFCx.ParameterSetName[7] := ' ';
   Line[19].DFCx.ParameterSetName[8] := ' ';
   Line[19].DFCx.ParameterSetName[9] := ' ';
   Line[19].DFCx.ParameterSetName[10] := ' ';
   Line[19].DFCx.ParameterSetName[11] := ' ';
   Line[19].DFCx.ParameterSetName[12] := ' ';
   Line[19].DFCx.ParameterSetName[13] := ' ';
   Line[19].DFCx.ParameterSetName[14] := ' ';
   Line[19].DFCx.ParameterSetName[15] := ' ';
   Line[19].DFCx.ParameterSetName[16] := ' ';
   Line[19].DFCx.ParameterSetName[17] := ' ';
   Line[19].DFCx.ParameterSetName[18] := ' ';
   Line[19].DFCx.ParameterSetName[19] := ' ';
   Line[19].DFCx.ParameterSetName[20] := ' ';
   Line[19].DFCx.ParameterSetName[21] := ' ';
   Line[19].DFCx.ParameterSetName[22] := ' ';
   Line[19].DFCx.ParameterSetName[23] := ' ';
   Line[19].DFCx.ParameterSetName[24] := ' ';
   Line[19].DFCx.ParameterSetName[25] := ' ';
   Line[19].DFCx.ParameterSetName[26] := ' ';
   Line[19].DFCx.ParameterSetName[27] := ' ';
   Line[19].DFCx.ParameterSetName[28] := ' ';
   Line[19].DFCx.ParameterSetName[29] := ' ';
   Line[19].DFCx.ParameterSetName[30] := ' ';
   Line[20].DFCx.PelletingDieName[1] := ' ';
   Line[20].DFCx.PelletingDieName[2] := ' ';
   Line[20].DFCx.PelletingDieName[3] := ' ';
   Line[20].DFCx.PelletingDieName[4] := ' ';
   Line[20].DFCx.PelletingDieName[5] := ' ';
   Line[20].DFCx.PelletingDieName[6] := ' ';
   Line[20].DFCx.PelletingDieName[7] := ' ';
   Line[20].DFCx.PelletingDieName[8] := ' ';
   Line[20].DFCx.PelletingDieName[9] := ' ';
   Line[20].DFCx.PelletingDieName[10] := ' ';
   Line[20].DFCx.ParameterSetIdent[1] := ' ';
   Line[20].DFCx.ParameterSetIdent[2] := ' ';
   Line[20].DFCx.ParameterSetIdent[3] := ' ';
   Line[20].DFCx.ParameterSetIdent[4] := ' ';
   Line[20].DFCx.ParameterSetIdent[5] := ' ';
   Line[20].DFCx.ParameterSetIdent[6] := ' ';
   Line[20].DFCx.ParameterSetIdent[7] := ' ';
   Line[20].DFCx.ParameterSetIdent[8] := ' ';
   Line[20].DFCx.ParameterSetIdent[9] := ' ';
   Line[20].DFCx.ParameterSetIdent[10] := ' ';
   Line[20].DFCx.ParameterSetIdent[11] := ' ';
   Line[20].DFCx.ParameterSetIdent[12] := ' ';
   Line[20].DFCx.ParameterSetIdent[13] := ' ';
   Line[20].DFCx.ParameterSetIdent[14] := ' ';
   Line[20].DFCx.ParameterSetIdent[15] := ' ';
   Line[20].DFCx.ParameterSetIdent[16] := ' ';
   Line[20].DFCx.ParameterSetName[1] := ' ';
   Line[20].DFCx.ParameterSetName[2] := ' ';
   Line[20].DFCx.ParameterSetName[3] := ' ';
   Line[20].DFCx.ParameterSetName[4] := ' ';
   Line[20].DFCx.ParameterSetName[5] := ' ';
   Line[20].DFCx.ParameterSetName[6] := ' ';
   Line[20].DFCx.ParameterSetName[7] := ' ';
   Line[20].DFCx.ParameterSetName[8] := ' ';
   Line[20].DFCx.ParameterSetName[9] := ' ';
   Line[20].DFCx.ParameterSetName[10] := ' ';
   Line[20].DFCx.ParameterSetName[11] := ' ';
   Line[20].DFCx.ParameterSetName[12] := ' ';
   Line[20].DFCx.ParameterSetName[13] := ' ';
   Line[20].DFCx.ParameterSetName[14] := ' ';
   Line[20].DFCx.ParameterSetName[15] := ' ';
   Line[20].DFCx.ParameterSetName[16] := ' ';
   Line[20].DFCx.ParameterSetName[17] := ' ';
   Line[20].DFCx.ParameterSetName[18] := ' ';
   Line[20].DFCx.ParameterSetName[19] := ' ';
   Line[20].DFCx.ParameterSetName[20] := ' ';
   Line[20].DFCx.ParameterSetName[21] := ' ';
   Line[20].DFCx.ParameterSetName[22] := ' ';
   Line[20].DFCx.ParameterSetName[23] := ' ';
   Line[20].DFCx.ParameterSetName[24] := ' ';
   Line[20].DFCx.ParameterSetName[25] := ' ';
   Line[20].DFCx.ParameterSetName[26] := ' ';
   Line[20].DFCx.ParameterSetName[27] := ' ';
   Line[20].DFCx.ParameterSetName[28] := ' ';
   Line[20].DFCx.ParameterSetName[29] := ' ';
   Line[20].DFCx.ParameterSetName[30] := ' ';
   Line[21].DFCx.PelletingDieName[1] := ' ';
   Line[21].DFCx.PelletingDieName[2] := ' ';
   Line[21].DFCx.PelletingDieName[3] := ' ';
   Line[21].DFCx.PelletingDieName[4] := ' ';
   Line[21].DFCx.PelletingDieName[5] := ' ';
   Line[21].DFCx.PelletingDieName[6] := ' ';
   Line[21].DFCx.PelletingDieName[7] := ' ';
   Line[21].DFCx.PelletingDieName[8] := ' ';
   Line[21].DFCx.PelletingDieName[9] := ' ';
   Line[21].DFCx.PelletingDieName[10] := ' ';
   Line[21].DFCx.ParameterSetIdent[1] := ' ';
   Line[21].DFCx.ParameterSetIdent[2] := ' ';
   Line[21].DFCx.ParameterSetIdent[3] := ' ';
   Line[21].DFCx.ParameterSetIdent[4] := ' ';
   Line[21].DFCx.ParameterSetIdent[5] := ' ';
   Line[21].DFCx.ParameterSetIdent[6] := ' ';
   Line[21].DFCx.ParameterSetIdent[7] := ' ';
   Line[21].DFCx.ParameterSetIdent[8] := ' ';
   Line[21].DFCx.ParameterSetIdent[9] := ' ';
   Line[21].DFCx.ParameterSetIdent[10] := ' ';
   Line[21].DFCx.ParameterSetIdent[11] := ' ';
   Line[21].DFCx.ParameterSetIdent[12] := ' ';
   Line[21].DFCx.ParameterSetIdent[13] := ' ';
   Line[21].DFCx.ParameterSetIdent[14] := ' ';
   Line[21].DFCx.ParameterSetIdent[15] := ' ';
   Line[21].DFCx.ParameterSetIdent[16] := ' ';
   Line[21].DFCx.ParameterSetName[1] := ' ';
   Line[21].DFCx.ParameterSetName[2] := ' ';
   Line[21].DFCx.ParameterSetName[3] := ' ';
   Line[21].DFCx.ParameterSetName[4] := ' ';
   Line[21].DFCx.ParameterSetName[5] := ' ';
   Line[21].DFCx.ParameterSetName[6] := ' ';
   Line[21].DFCx.ParameterSetName[7] := ' ';
   Line[21].DFCx.ParameterSetName[8] := ' ';
   Line[21].DFCx.ParameterSetName[9] := ' ';
   Line[21].DFCx.ParameterSetName[10] := ' ';
   Line[21].DFCx.ParameterSetName[11] := ' ';
   Line[21].DFCx.ParameterSetName[12] := ' ';
   Line[21].DFCx.ParameterSetName[13] := ' ';
   Line[21].DFCx.ParameterSetName[14] := ' ';
   Line[21].DFCx.ParameterSetName[15] := ' ';
   Line[21].DFCx.ParameterSetName[16] := ' ';
   Line[21].DFCx.ParameterSetName[17] := ' ';
   Line[21].DFCx.ParameterSetName[18] := ' ';
   Line[21].DFCx.ParameterSetName[19] := ' ';
   Line[21].DFCx.ParameterSetName[20] := ' ';
   Line[21].DFCx.ParameterSetName[21] := ' ';
   Line[21].DFCx.ParameterSetName[22] := ' ';
   Line[21].DFCx.ParameterSetName[23] := ' ';
   Line[21].DFCx.ParameterSetName[24] := ' ';
   Line[21].DFCx.ParameterSetName[25] := ' ';
   Line[21].DFCx.ParameterSetName[26] := ' ';
   Line[21].DFCx.ParameterSetName[27] := ' ';
   Line[21].DFCx.ParameterSetName[28] := ' ';
   Line[21].DFCx.ParameterSetName[29] := ' ';
   Line[21].DFCx.ParameterSetName[30] := ' ';
   Line[22].DFCx.PelletingDieName[1] := ' ';
   Line[22].DFCx.PelletingDieName[2] := ' ';
   Line[22].DFCx.PelletingDieName[3] := ' ';
   Line[22].DFCx.PelletingDieName[4] := ' ';
   Line[22].DFCx.PelletingDieName[5] := ' ';
   Line[22].DFCx.PelletingDieName[6] := ' ';
   Line[22].DFCx.PelletingDieName[7] := ' ';
   Line[22].DFCx.PelletingDieName[8] := ' ';
   Line[22].DFCx.PelletingDieName[9] := ' ';
   Line[22].DFCx.PelletingDieName[10] := ' ';
   Line[22].DFCx.ParameterSetIdent[1] := ' ';
   Line[22].DFCx.ParameterSetIdent[2] := ' ';
   Line[22].DFCx.ParameterSetIdent[3] := ' ';
   Line[22].DFCx.ParameterSetIdent[4] := ' ';
   Line[22].DFCx.ParameterSetIdent[5] := ' ';
   Line[22].DFCx.ParameterSetIdent[6] := ' ';
   Line[22].DFCx.ParameterSetIdent[7] := ' ';
   Line[22].DFCx.ParameterSetIdent[8] := ' ';
   Line[22].DFCx.ParameterSetIdent[9] := ' ';
   Line[22].DFCx.ParameterSetIdent[10] := ' ';
   Line[22].DFCx.ParameterSetIdent[11] := ' ';
   Line[22].DFCx.ParameterSetIdent[12] := ' ';
   Line[22].DFCx.ParameterSetIdent[13] := ' ';
   Line[22].DFCx.ParameterSetIdent[14] := ' ';
   Line[22].DFCx.ParameterSetIdent[15] := ' ';
   Line[22].DFCx.ParameterSetIdent[16] := ' ';
   Line[22].DFCx.ParameterSetName[1] := ' ';
   Line[22].DFCx.ParameterSetName[2] := ' ';
   Line[22].DFCx.ParameterSetName[3] := ' ';
   Line[22].DFCx.ParameterSetName[4] := ' ';
   Line[22].DFCx.ParameterSetName[5] := ' ';
   Line[22].DFCx.ParameterSetName[6] := ' ';
   Line[22].DFCx.ParameterSetName[7] := ' ';
   Line[22].DFCx.ParameterSetName[8] := ' ';
   Line[22].DFCx.ParameterSetName[9] := ' ';
   Line[22].DFCx.ParameterSetName[10] := ' ';
   Line[22].DFCx.ParameterSetName[11] := ' ';
   Line[22].DFCx.ParameterSetName[12] := ' ';
   Line[22].DFCx.ParameterSetName[13] := ' ';
   Line[22].DFCx.ParameterSetName[14] := ' ';
   Line[22].DFCx.ParameterSetName[15] := ' ';
   Line[22].DFCx.ParameterSetName[16] := ' ';
   Line[22].DFCx.ParameterSetName[17] := ' ';
   Line[22].DFCx.ParameterSetName[18] := ' ';
   Line[22].DFCx.ParameterSetName[19] := ' ';
   Line[22].DFCx.ParameterSetName[20] := ' ';
   Line[22].DFCx.ParameterSetName[21] := ' ';
   Line[22].DFCx.ParameterSetName[22] := ' ';
   Line[22].DFCx.ParameterSetName[23] := ' ';
   Line[22].DFCx.ParameterSetName[24] := ' ';
   Line[22].DFCx.ParameterSetName[25] := ' ';
   Line[22].DFCx.ParameterSetName[26] := ' ';
   Line[22].DFCx.ParameterSetName[27] := ' ';
   Line[22].DFCx.ParameterSetName[28] := ' ';
   Line[22].DFCx.ParameterSetName[29] := ' ';
   Line[22].DFCx.ParameterSetName[30] := ' ';
   Line[23].DFCx.PelletingDieName[1] := ' ';
   Line[23].DFCx.PelletingDieName[2] := ' ';
   Line[23].DFCx.PelletingDieName[3] := ' ';
   Line[23].DFCx.PelletingDieName[4] := ' ';
   Line[23].DFCx.PelletingDieName[5] := ' ';
   Line[23].DFCx.PelletingDieName[6] := ' ';
   Line[23].DFCx.PelletingDieName[7] := ' ';
   Line[23].DFCx.PelletingDieName[8] := ' ';
   Line[23].DFCx.PelletingDieName[9] := ' ';
   Line[23].DFCx.PelletingDieName[10] := ' ';
   Line[23].DFCx.ParameterSetIdent[1] := ' ';
   Line[23].DFCx.ParameterSetIdent[2] := ' ';
   Line[23].DFCx.ParameterSetIdent[3] := ' ';
   Line[23].DFCx.ParameterSetIdent[4] := ' ';
   Line[23].DFCx.ParameterSetIdent[5] := ' ';
   Line[23].DFCx.ParameterSetIdent[6] := ' ';
   Line[23].DFCx.ParameterSetIdent[7] := ' ';
   Line[23].DFCx.ParameterSetIdent[8] := ' ';
   Line[23].DFCx.ParameterSetIdent[9] := ' ';
   Line[23].DFCx.ParameterSetIdent[10] := ' ';
   Line[23].DFCx.ParameterSetIdent[11] := ' ';
   Line[23].DFCx.ParameterSetIdent[12] := ' ';
   Line[23].DFCx.ParameterSetIdent[13] := ' ';
   Line[23].DFCx.ParameterSetIdent[14] := ' ';
   Line[23].DFCx.ParameterSetIdent[15] := ' ';
   Line[23].DFCx.ParameterSetIdent[16] := ' ';
   Line[23].DFCx.ParameterSetName[1] := ' ';
   Line[23].DFCx.ParameterSetName[2] := ' ';
   Line[23].DFCx.ParameterSetName[3] := ' ';
   Line[23].DFCx.ParameterSetName[4] := ' ';
   Line[23].DFCx.ParameterSetName[5] := ' ';
   Line[23].DFCx.ParameterSetName[6] := ' ';
   Line[23].DFCx.ParameterSetName[7] := ' ';
   Line[23].DFCx.ParameterSetName[8] := ' ';
   Line[23].DFCx.ParameterSetName[9] := ' ';
   Line[23].DFCx.ParameterSetName[10] := ' ';
   Line[23].DFCx.ParameterSetName[11] := ' ';
   Line[23].DFCx.ParameterSetName[12] := ' ';
   Line[23].DFCx.ParameterSetName[13] := ' ';
   Line[23].DFCx.ParameterSetName[14] := ' ';
   Line[23].DFCx.ParameterSetName[15] := ' ';
   Line[23].DFCx.ParameterSetName[16] := ' ';
   Line[23].DFCx.ParameterSetName[17] := ' ';
   Line[23].DFCx.ParameterSetName[18] := ' ';
   Line[23].DFCx.ParameterSetName[19] := ' ';
   Line[23].DFCx.ParameterSetName[20] := ' ';
   Line[23].DFCx.ParameterSetName[21] := ' ';
   Line[23].DFCx.ParameterSetName[22] := ' ';
   Line[23].DFCx.ParameterSetName[23] := ' ';
   Line[23].DFCx.ParameterSetName[24] := ' ';
   Line[23].DFCx.ParameterSetName[25] := ' ';
   Line[23].DFCx.ParameterSetName[26] := ' ';
   Line[23].DFCx.ParameterSetName[27] := ' ';
   Line[23].DFCx.ParameterSetName[28] := ' ';
   Line[23].DFCx.ParameterSetName[29] := ' ';
   Line[23].DFCx.ParameterSetName[30] := ' ';
   Line[24].DFCx.PelletingDieName[1] := ' ';
   Line[24].DFCx.PelletingDieName[2] := ' ';
   Line[24].DFCx.PelletingDieName[3] := ' ';
   Line[24].DFCx.PelletingDieName[4] := ' ';
   Line[24].DFCx.PelletingDieName[5] := ' ';
   Line[24].DFCx.PelletingDieName[6] := ' ';
   Line[24].DFCx.PelletingDieName[7] := ' ';
   Line[24].DFCx.PelletingDieName[8] := ' ';
   Line[24].DFCx.PelletingDieName[9] := ' ';
   Line[24].DFCx.PelletingDieName[10] := ' ';
   Line[24].DFCx.ParameterSetIdent[1] := ' ';
   Line[24].DFCx.ParameterSetIdent[2] := ' ';
   Line[24].DFCx.ParameterSetIdent[3] := ' ';
   Line[24].DFCx.ParameterSetIdent[4] := ' ';
   Line[24].DFCx.ParameterSetIdent[5] := ' ';
   Line[24].DFCx.ParameterSetIdent[6] := ' ';
   Line[24].DFCx.ParameterSetIdent[7] := ' ';
   Line[24].DFCx.ParameterSetIdent[8] := ' ';
   Line[24].DFCx.ParameterSetIdent[9] := ' ';
   Line[24].DFCx.ParameterSetIdent[10] := ' ';
   Line[24].DFCx.ParameterSetIdent[11] := ' ';
   Line[24].DFCx.ParameterSetIdent[12] := ' ';
   Line[24].DFCx.ParameterSetIdent[13] := ' ';
   Line[24].DFCx.ParameterSetIdent[14] := ' ';
   Line[24].DFCx.ParameterSetIdent[15] := ' ';
   Line[24].DFCx.ParameterSetIdent[16] := ' ';
   Line[24].DFCx.ParameterSetName[1] := ' ';
   Line[24].DFCx.ParameterSetName[2] := ' ';
   Line[24].DFCx.ParameterSetName[3] := ' ';
   Line[24].DFCx.ParameterSetName[4] := ' ';
   Line[24].DFCx.ParameterSetName[5] := ' ';
   Line[24].DFCx.ParameterSetName[6] := ' ';
   Line[24].DFCx.ParameterSetName[7] := ' ';
   Line[24].DFCx.ParameterSetName[8] := ' ';
   Line[24].DFCx.ParameterSetName[9] := ' ';
   Line[24].DFCx.ParameterSetName[10] := ' ';
   Line[24].DFCx.ParameterSetName[11] := ' ';
   Line[24].DFCx.ParameterSetName[12] := ' ';
   Line[24].DFCx.ParameterSetName[13] := ' ';
   Line[24].DFCx.ParameterSetName[14] := ' ';
   Line[24].DFCx.ParameterSetName[15] := ' ';
   Line[24].DFCx.ParameterSetName[16] := ' ';
   Line[24].DFCx.ParameterSetName[17] := ' ';
   Line[24].DFCx.ParameterSetName[18] := ' ';
   Line[24].DFCx.ParameterSetName[19] := ' ';
   Line[24].DFCx.ParameterSetName[20] := ' ';
   Line[24].DFCx.ParameterSetName[21] := ' ';
   Line[24].DFCx.ParameterSetName[22] := ' ';
   Line[24].DFCx.ParameterSetName[23] := ' ';
   Line[24].DFCx.ParameterSetName[24] := ' ';
   Line[24].DFCx.ParameterSetName[25] := ' ';
   Line[24].DFCx.ParameterSetName[26] := ' ';
   Line[24].DFCx.ParameterSetName[27] := ' ';
   Line[24].DFCx.ParameterSetName[28] := ' ';
   Line[24].DFCx.ParameterSetName[29] := ' ';
   Line[24].DFCx.ParameterSetName[30] := ' ';
   Line[25].DFCx.PelletingDieName[1] := ' ';
   Line[25].DFCx.PelletingDieName[2] := ' ';
   Line[25].DFCx.PelletingDieName[3] := ' ';
   Line[25].DFCx.PelletingDieName[4] := ' ';
   Line[25].DFCx.PelletingDieName[5] := ' ';
   Line[25].DFCx.PelletingDieName[6] := ' ';
   Line[25].DFCx.PelletingDieName[7] := ' ';
   Line[25].DFCx.PelletingDieName[8] := ' ';
   Line[25].DFCx.PelletingDieName[9] := ' ';
   Line[25].DFCx.PelletingDieName[10] := ' ';
   Line[25].DFCx.ParameterSetIdent[1] := ' ';
   Line[25].DFCx.ParameterSetIdent[2] := ' ';
   Line[25].DFCx.ParameterSetIdent[3] := ' ';
   Line[25].DFCx.ParameterSetIdent[4] := ' ';
   Line[25].DFCx.ParameterSetIdent[5] := ' ';
   Line[25].DFCx.ParameterSetIdent[6] := ' ';
   Line[25].DFCx.ParameterSetIdent[7] := ' ';
   Line[25].DFCx.ParameterSetIdent[8] := ' ';
   Line[25].DFCx.ParameterSetIdent[9] := ' ';
   Line[25].DFCx.ParameterSetIdent[10] := ' ';
   Line[25].DFCx.ParameterSetIdent[11] := ' ';
   Line[25].DFCx.ParameterSetIdent[12] := ' ';
   Line[25].DFCx.ParameterSetIdent[13] := ' ';
   Line[25].DFCx.ParameterSetIdent[14] := ' ';
   Line[25].DFCx.ParameterSetIdent[15] := ' ';
   Line[25].DFCx.ParameterSetIdent[16] := ' ';
   Line[25].DFCx.ParameterSetName[1] := ' ';
   Line[25].DFCx.ParameterSetName[2] := ' ';
   Line[25].DFCx.ParameterSetName[3] := ' ';
   Line[25].DFCx.ParameterSetName[4] := ' ';
   Line[25].DFCx.ParameterSetName[5] := ' ';
   Line[25].DFCx.ParameterSetName[6] := ' ';
   Line[25].DFCx.ParameterSetName[7] := ' ';
   Line[25].DFCx.ParameterSetName[8] := ' ';
   Line[25].DFCx.ParameterSetName[9] := ' ';
   Line[25].DFCx.ParameterSetName[10] := ' ';
   Line[25].DFCx.ParameterSetName[11] := ' ';
   Line[25].DFCx.ParameterSetName[12] := ' ';
   Line[25].DFCx.ParameterSetName[13] := ' ';
   Line[25].DFCx.ParameterSetName[14] := ' ';
   Line[25].DFCx.ParameterSetName[15] := ' ';
   Line[25].DFCx.ParameterSetName[16] := ' ';
   Line[25].DFCx.ParameterSetName[17] := ' ';
   Line[25].DFCx.ParameterSetName[18] := ' ';
   Line[25].DFCx.ParameterSetName[19] := ' ';
   Line[25].DFCx.ParameterSetName[20] := ' ';
   Line[25].DFCx.ParameterSetName[21] := ' ';
   Line[25].DFCx.ParameterSetName[22] := ' ';
   Line[25].DFCx.ParameterSetName[23] := ' ';
   Line[25].DFCx.ParameterSetName[24] := ' ';
   Line[25].DFCx.ParameterSetName[25] := ' ';
   Line[25].DFCx.ParameterSetName[26] := ' ';
   Line[25].DFCx.ParameterSetName[27] := ' ';
   Line[25].DFCx.ParameterSetName[28] := ' ';
   Line[25].DFCx.ParameterSetName[29] := ' ';
   Line[25].DFCx.ParameterSetName[30] := ' ';
   Line[26].DFCx.PelletingDieName[1] := ' ';
   Line[26].DFCx.PelletingDieName[2] := ' ';
   Line[26].DFCx.PelletingDieName[3] := ' ';
   Line[26].DFCx.PelletingDieName[4] := ' ';
   Line[26].DFCx.PelletingDieName[5] := ' ';
   Line[26].DFCx.PelletingDieName[6] := ' ';
   Line[26].DFCx.PelletingDieName[7] := ' ';
   Line[26].DFCx.PelletingDieName[8] := ' ';
   Line[26].DFCx.PelletingDieName[9] := ' ';
   Line[26].DFCx.PelletingDieName[10] := ' ';
   Line[26].DFCx.ParameterSetIdent[1] := ' ';
   Line[26].DFCx.ParameterSetIdent[2] := ' ';
   Line[26].DFCx.ParameterSetIdent[3] := ' ';
   Line[26].DFCx.ParameterSetIdent[4] := ' ';
   Line[26].DFCx.ParameterSetIdent[5] := ' ';
   Line[26].DFCx.ParameterSetIdent[6] := ' ';
   Line[26].DFCx.ParameterSetIdent[7] := ' ';
   Line[26].DFCx.ParameterSetIdent[8] := ' ';
   Line[26].DFCx.ParameterSetIdent[9] := ' ';
   Line[26].DFCx.ParameterSetIdent[10] := ' ';
   Line[26].DFCx.ParameterSetIdent[11] := ' ';
   Line[26].DFCx.ParameterSetIdent[12] := ' ';
   Line[26].DFCx.ParameterSetIdent[13] := ' ';
   Line[26].DFCx.ParameterSetIdent[14] := ' ';
   Line[26].DFCx.ParameterSetIdent[15] := ' ';
   Line[26].DFCx.ParameterSetIdent[16] := ' ';
   Line[26].DFCx.ParameterSetName[1] := ' ';
   Line[26].DFCx.ParameterSetName[2] := ' ';
   Line[26].DFCx.ParameterSetName[3] := ' ';
   Line[26].DFCx.ParameterSetName[4] := ' ';
   Line[26].DFCx.ParameterSetName[5] := ' ';
   Line[26].DFCx.ParameterSetName[6] := ' ';
   Line[26].DFCx.ParameterSetName[7] := ' ';
   Line[26].DFCx.ParameterSetName[8] := ' ';
   Line[26].DFCx.ParameterSetName[9] := ' ';
   Line[26].DFCx.ParameterSetName[10] := ' ';
   Line[26].DFCx.ParameterSetName[11] := ' ';
   Line[26].DFCx.ParameterSetName[12] := ' ';
   Line[26].DFCx.ParameterSetName[13] := ' ';
   Line[26].DFCx.ParameterSetName[14] := ' ';
   Line[26].DFCx.ParameterSetName[15] := ' ';
   Line[26].DFCx.ParameterSetName[16] := ' ';
   Line[26].DFCx.ParameterSetName[17] := ' ';
   Line[26].DFCx.ParameterSetName[18] := ' ';
   Line[26].DFCx.ParameterSetName[19] := ' ';
   Line[26].DFCx.ParameterSetName[20] := ' ';
   Line[26].DFCx.ParameterSetName[21] := ' ';
   Line[26].DFCx.ParameterSetName[22] := ' ';
   Line[26].DFCx.ParameterSetName[23] := ' ';
   Line[26].DFCx.ParameterSetName[24] := ' ';
   Line[26].DFCx.ParameterSetName[25] := ' ';
   Line[26].DFCx.ParameterSetName[26] := ' ';
   Line[26].DFCx.ParameterSetName[27] := ' ';
   Line[26].DFCx.ParameterSetName[28] := ' ';
   Line[26].DFCx.ParameterSetName[29] := ' ';
   Line[26].DFCx.ParameterSetName[30] := ' ';
   Line[27].DFCx.PelletingDieName[1] := ' ';
   Line[27].DFCx.PelletingDieName[2] := ' ';
   Line[27].DFCx.PelletingDieName[3] := ' ';
   Line[27].DFCx.PelletingDieName[4] := ' ';
   Line[27].DFCx.PelletingDieName[5] := ' ';
   Line[27].DFCx.PelletingDieName[6] := ' ';
   Line[27].DFCx.PelletingDieName[7] := ' ';
   Line[27].DFCx.PelletingDieName[8] := ' ';
   Line[27].DFCx.PelletingDieName[9] := ' ';
   Line[27].DFCx.PelletingDieName[10] := ' ';
   Line[27].DFCx.ParameterSetIdent[1] := ' ';
   Line[27].DFCx.ParameterSetIdent[2] := ' ';
   Line[27].DFCx.ParameterSetIdent[3] := ' ';
   Line[27].DFCx.ParameterSetIdent[4] := ' ';
   Line[27].DFCx.ParameterSetIdent[5] := ' ';
   Line[27].DFCx.ParameterSetIdent[6] := ' ';
   Line[27].DFCx.ParameterSetIdent[7] := ' ';
   Line[27].DFCx.ParameterSetIdent[8] := ' ';
   Line[27].DFCx.ParameterSetIdent[9] := ' ';
   Line[27].DFCx.ParameterSetIdent[10] := ' ';
   Line[27].DFCx.ParameterSetIdent[11] := ' ';
   Line[27].DFCx.ParameterSetIdent[12] := ' ';
   Line[27].DFCx.ParameterSetIdent[13] := ' ';
   Line[27].DFCx.ParameterSetIdent[14] := ' ';
   Line[27].DFCx.ParameterSetIdent[15] := ' ';
   Line[27].DFCx.ParameterSetIdent[16] := ' ';
   Line[27].DFCx.ParameterSetName[1] := ' ';
   Line[27].DFCx.ParameterSetName[2] := ' ';
   Line[27].DFCx.ParameterSetName[3] := ' ';
   Line[27].DFCx.ParameterSetName[4] := ' ';
   Line[27].DFCx.ParameterSetName[5] := ' ';
   Line[27].DFCx.ParameterSetName[6] := ' ';
   Line[27].DFCx.ParameterSetName[7] := ' ';
   Line[27].DFCx.ParameterSetName[8] := ' ';
   Line[27].DFCx.ParameterSetName[9] := ' ';
   Line[27].DFCx.ParameterSetName[10] := ' ';
   Line[27].DFCx.ParameterSetName[11] := ' ';
   Line[27].DFCx.ParameterSetName[12] := ' ';
   Line[27].DFCx.ParameterSetName[13] := ' ';
   Line[27].DFCx.ParameterSetName[14] := ' ';
   Line[27].DFCx.ParameterSetName[15] := ' ';
   Line[27].DFCx.ParameterSetName[16] := ' ';
   Line[27].DFCx.ParameterSetName[17] := ' ';
   Line[27].DFCx.ParameterSetName[18] := ' ';
   Line[27].DFCx.ParameterSetName[19] := ' ';
   Line[27].DFCx.ParameterSetName[20] := ' ';
   Line[27].DFCx.ParameterSetName[21] := ' ';
   Line[27].DFCx.ParameterSetName[22] := ' ';
   Line[27].DFCx.ParameterSetName[23] := ' ';
   Line[27].DFCx.ParameterSetName[24] := ' ';
   Line[27].DFCx.ParameterSetName[25] := ' ';
   Line[27].DFCx.ParameterSetName[26] := ' ';
   Line[27].DFCx.ParameterSetName[27] := ' ';
   Line[27].DFCx.ParameterSetName[28] := ' ';
   Line[27].DFCx.ParameterSetName[29] := ' ';
   Line[27].DFCx.ParameterSetName[30] := ' ';
   Line[28].DFCx.PelletingDieName[1] := ' ';
   Line[28].DFCx.PelletingDieName[2] := ' ';
   Line[28].DFCx.PelletingDieName[3] := ' ';
   Line[28].DFCx.PelletingDieName[4] := ' ';
   Line[28].DFCx.PelletingDieName[5] := ' ';
   Line[28].DFCx.PelletingDieName[6] := ' ';
   Line[28].DFCx.PelletingDieName[7] := ' ';
   Line[28].DFCx.PelletingDieName[8] := ' ';
   Line[28].DFCx.PelletingDieName[9] := ' ';
   Line[28].DFCx.PelletingDieName[10] := ' ';
   Line[28].DFCx.ParameterSetIdent[1] := ' ';
   Line[28].DFCx.ParameterSetIdent[2] := ' ';
   Line[28].DFCx.ParameterSetIdent[3] := ' ';
   Line[28].DFCx.ParameterSetIdent[4] := ' ';
   Line[28].DFCx.ParameterSetIdent[5] := ' ';
   Line[28].DFCx.ParameterSetIdent[6] := ' ';
   Line[28].DFCx.ParameterSetIdent[7] := ' ';
   Line[28].DFCx.ParameterSetIdent[8] := ' ';
   Line[28].DFCx.ParameterSetIdent[9] := ' ';
   Line[28].DFCx.ParameterSetIdent[10] := ' ';
   Line[28].DFCx.ParameterSetIdent[11] := ' ';
   Line[28].DFCx.ParameterSetIdent[12] := ' ';
   Line[28].DFCx.ParameterSetIdent[13] := ' ';
   Line[28].DFCx.ParameterSetIdent[14] := ' ';
   Line[28].DFCx.ParameterSetIdent[15] := ' ';
   Line[28].DFCx.ParameterSetIdent[16] := ' ';
   Line[28].DFCx.ParameterSetName[1] := ' ';
   Line[28].DFCx.ParameterSetName[2] := ' ';
   Line[28].DFCx.ParameterSetName[3] := ' ';
   Line[28].DFCx.ParameterSetName[4] := ' ';
   Line[28].DFCx.ParameterSetName[5] := ' ';
   Line[28].DFCx.ParameterSetName[6] := ' ';
   Line[28].DFCx.ParameterSetName[7] := ' ';
   Line[28].DFCx.ParameterSetName[8] := ' ';
   Line[28].DFCx.ParameterSetName[9] := ' ';
   Line[28].DFCx.ParameterSetName[10] := ' ';
   Line[28].DFCx.ParameterSetName[11] := ' ';
   Line[28].DFCx.ParameterSetName[12] := ' ';
   Line[28].DFCx.ParameterSetName[13] := ' ';
   Line[28].DFCx.ParameterSetName[14] := ' ';
   Line[28].DFCx.ParameterSetName[15] := ' ';
   Line[28].DFCx.ParameterSetName[16] := ' ';
   Line[28].DFCx.ParameterSetName[17] := ' ';
   Line[28].DFCx.ParameterSetName[18] := ' ';
   Line[28].DFCx.ParameterSetName[19] := ' ';
   Line[28].DFCx.ParameterSetName[20] := ' ';
   Line[28].DFCx.ParameterSetName[21] := ' ';
   Line[28].DFCx.ParameterSetName[22] := ' ';
   Line[28].DFCx.ParameterSetName[23] := ' ';
   Line[28].DFCx.ParameterSetName[24] := ' ';
   Line[28].DFCx.ParameterSetName[25] := ' ';
   Line[28].DFCx.ParameterSetName[26] := ' ';
   Line[28].DFCx.ParameterSetName[27] := ' ';
   Line[28].DFCx.ParameterSetName[28] := ' ';
   Line[28].DFCx.ParameterSetName[29] := ' ';
   Line[28].DFCx.ParameterSetName[30] := ' ';
   Line[29].DFCx.PelletingDieName[1] := ' ';
   Line[29].DFCx.PelletingDieName[2] := ' ';
   Line[29].DFCx.PelletingDieName[3] := ' ';
   Line[29].DFCx.PelletingDieName[4] := ' ';
   Line[29].DFCx.PelletingDieName[5] := ' ';
   Line[29].DFCx.PelletingDieName[6] := ' ';
   Line[29].DFCx.PelletingDieName[7] := ' ';
   Line[29].DFCx.PelletingDieName[8] := ' ';
   Line[29].DFCx.PelletingDieName[9] := ' ';
   Line[29].DFCx.PelletingDieName[10] := ' ';
   Line[29].DFCx.ParameterSetIdent[1] := ' ';
   Line[29].DFCx.ParameterSetIdent[2] := ' ';
   Line[29].DFCx.ParameterSetIdent[3] := ' ';
   Line[29].DFCx.ParameterSetIdent[4] := ' ';
   Line[29].DFCx.ParameterSetIdent[5] := ' ';
   Line[29].DFCx.ParameterSetIdent[6] := ' ';
   Line[29].DFCx.ParameterSetIdent[7] := ' ';
   Line[29].DFCx.ParameterSetIdent[8] := ' ';
   Line[29].DFCx.ParameterSetIdent[9] := ' ';
   Line[29].DFCx.ParameterSetIdent[10] := ' ';
   Line[29].DFCx.ParameterSetIdent[11] := ' ';
   Line[29].DFCx.ParameterSetIdent[12] := ' ';
   Line[29].DFCx.ParameterSetIdent[13] := ' ';
   Line[29].DFCx.ParameterSetIdent[14] := ' ';
   Line[29].DFCx.ParameterSetIdent[15] := ' ';
   Line[29].DFCx.ParameterSetIdent[16] := ' ';
   Line[29].DFCx.ParameterSetName[1] := ' ';
   Line[29].DFCx.ParameterSetName[2] := ' ';
   Line[29].DFCx.ParameterSetName[3] := ' ';
   Line[29].DFCx.ParameterSetName[4] := ' ';
   Line[29].DFCx.ParameterSetName[5] := ' ';
   Line[29].DFCx.ParameterSetName[6] := ' ';
   Line[29].DFCx.ParameterSetName[7] := ' ';
   Line[29].DFCx.ParameterSetName[8] := ' ';
   Line[29].DFCx.ParameterSetName[9] := ' ';
   Line[29].DFCx.ParameterSetName[10] := ' ';
   Line[29].DFCx.ParameterSetName[11] := ' ';
   Line[29].DFCx.ParameterSetName[12] := ' ';
   Line[29].DFCx.ParameterSetName[13] := ' ';
   Line[29].DFCx.ParameterSetName[14] := ' ';
   Line[29].DFCx.ParameterSetName[15] := ' ';
   Line[29].DFCx.ParameterSetName[16] := ' ';
   Line[29].DFCx.ParameterSetName[17] := ' ';
   Line[29].DFCx.ParameterSetName[18] := ' ';
   Line[29].DFCx.ParameterSetName[19] := ' ';
   Line[29].DFCx.ParameterSetName[20] := ' ';
   Line[29].DFCx.ParameterSetName[21] := ' ';
   Line[29].DFCx.ParameterSetName[22] := ' ';
   Line[29].DFCx.ParameterSetName[23] := ' ';
   Line[29].DFCx.ParameterSetName[24] := ' ';
   Line[29].DFCx.ParameterSetName[25] := ' ';
   Line[29].DFCx.ParameterSetName[26] := ' ';
   Line[29].DFCx.ParameterSetName[27] := ' ';
   Line[29].DFCx.ParameterSetName[28] := ' ';
   Line[29].DFCx.ParameterSetName[29] := ' ';
   Line[29].DFCx.ParameterSetName[30] := ' ';
   Line[30].DFCx.PelletingDieName[1] := ' ';
   Line[30].DFCx.PelletingDieName[2] := ' ';
   Line[30].DFCx.PelletingDieName[3] := ' ';
   Line[30].DFCx.PelletingDieName[4] := ' ';
   Line[30].DFCx.PelletingDieName[5] := ' ';
   Line[30].DFCx.PelletingDieName[6] := ' ';
   Line[30].DFCx.PelletingDieName[7] := ' ';
   Line[30].DFCx.PelletingDieName[8] := ' ';
   Line[30].DFCx.PelletingDieName[9] := ' ';
   Line[30].DFCx.PelletingDieName[10] := ' ';
   Line[30].DFCx.ParameterSetIdent[1] := ' ';
   Line[30].DFCx.ParameterSetIdent[2] := ' ';
   Line[30].DFCx.ParameterSetIdent[3] := ' ';
   Line[30].DFCx.ParameterSetIdent[4] := ' ';
   Line[30].DFCx.ParameterSetIdent[5] := ' ';
   Line[30].DFCx.ParameterSetIdent[6] := ' ';
   Line[30].DFCx.ParameterSetIdent[7] := ' ';
   Line[30].DFCx.ParameterSetIdent[8] := ' ';
   Line[30].DFCx.ParameterSetIdent[9] := ' ';
   Line[30].DFCx.ParameterSetIdent[10] := ' ';
   Line[30].DFCx.ParameterSetIdent[11] := ' ';
   Line[30].DFCx.ParameterSetIdent[12] := ' ';
   Line[30].DFCx.ParameterSetIdent[13] := ' ';
   Line[30].DFCx.ParameterSetIdent[14] := ' ';
   Line[30].DFCx.ParameterSetIdent[15] := ' ';
   Line[30].DFCx.ParameterSetIdent[16] := ' ';
   Line[30].DFCx.ParameterSetName[1] := ' ';
   Line[30].DFCx.ParameterSetName[2] := ' ';
   Line[30].DFCx.ParameterSetName[3] := ' ';
   Line[30].DFCx.ParameterSetName[4] := ' ';
   Line[30].DFCx.ParameterSetName[5] := ' ';
   Line[30].DFCx.ParameterSetName[6] := ' ';
   Line[30].DFCx.ParameterSetName[7] := ' ';
   Line[30].DFCx.ParameterSetName[8] := ' ';
   Line[30].DFCx.ParameterSetName[9] := ' ';
   Line[30].DFCx.ParameterSetName[10] := ' ';
   Line[30].DFCx.ParameterSetName[11] := ' ';
   Line[30].DFCx.ParameterSetName[12] := ' ';
   Line[30].DFCx.ParameterSetName[13] := ' ';
   Line[30].DFCx.ParameterSetName[14] := ' ';
   Line[30].DFCx.ParameterSetName[15] := ' ';
   Line[30].DFCx.ParameterSetName[16] := ' ';
   Line[30].DFCx.ParameterSetName[17] := ' ';
   Line[30].DFCx.ParameterSetName[18] := ' ';
   Line[30].DFCx.ParameterSetName[19] := ' ';
   Line[30].DFCx.ParameterSetName[20] := ' ';
   Line[30].DFCx.ParameterSetName[21] := ' ';
   Line[30].DFCx.ParameterSetName[22] := ' ';
   Line[30].DFCx.ParameterSetName[23] := ' ';
   Line[30].DFCx.ParameterSetName[24] := ' ';
   Line[30].DFCx.ParameterSetName[25] := ' ';
   Line[30].DFCx.ParameterSetName[26] := ' ';
   Line[30].DFCx.ParameterSetName[27] := ' ';
   Line[30].DFCx.ParameterSetName[28] := ' ';
   Line[30].DFCx.ParameterSetName[29] := ' ';
   Line[30].DFCx.ParameterSetName[30] := ' ';
   Line[31].DFCx.PelletingDieName[1] := ' ';
   Line[31].DFCx.PelletingDieName[2] := ' ';
   Line[31].DFCx.PelletingDieName[3] := ' ';
   Line[31].DFCx.PelletingDieName[4] := ' ';
   Line[31].DFCx.PelletingDieName[5] := ' ';
   Line[31].DFCx.PelletingDieName[6] := ' ';
   Line[31].DFCx.PelletingDieName[7] := ' ';
   Line[31].DFCx.PelletingDieName[8] := ' ';
   Line[31].DFCx.PelletingDieName[9] := ' ';
   Line[31].DFCx.PelletingDieName[10] := ' ';
   Line[31].DFCx.ParameterSetIdent[1] := ' ';
   Line[31].DFCx.ParameterSetIdent[2] := ' ';
   Line[31].DFCx.ParameterSetIdent[3] := ' ';
   Line[31].DFCx.ParameterSetIdent[4] := ' ';
   Line[31].DFCx.ParameterSetIdent[5] := ' ';
   Line[31].DFCx.ParameterSetIdent[6] := ' ';
   Line[31].DFCx.ParameterSetIdent[7] := ' ';
   Line[31].DFCx.ParameterSetIdent[8] := ' ';
   Line[31].DFCx.ParameterSetIdent[9] := ' ';
   Line[31].DFCx.ParameterSetIdent[10] := ' ';
   Line[31].DFCx.ParameterSetIdent[11] := ' ';
   Line[31].DFCx.ParameterSetIdent[12] := ' ';
   Line[31].DFCx.ParameterSetIdent[13] := ' ';
   Line[31].DFCx.ParameterSetIdent[14] := ' ';
   Line[31].DFCx.ParameterSetIdent[15] := ' ';
   Line[31].DFCx.ParameterSetIdent[16] := ' ';
   Line[31].DFCx.ParameterSetName[1] := ' ';
   Line[31].DFCx.ParameterSetName[2] := ' ';
   Line[31].DFCx.ParameterSetName[3] := ' ';
   Line[31].DFCx.ParameterSetName[4] := ' ';
   Line[31].DFCx.ParameterSetName[5] := ' ';
   Line[31].DFCx.ParameterSetName[6] := ' ';
   Line[31].DFCx.ParameterSetName[7] := ' ';
   Line[31].DFCx.ParameterSetName[8] := ' ';
   Line[31].DFCx.ParameterSetName[9] := ' ';
   Line[31].DFCx.ParameterSetName[10] := ' ';
   Line[31].DFCx.ParameterSetName[11] := ' ';
   Line[31].DFCx.ParameterSetName[12] := ' ';
   Line[31].DFCx.ParameterSetName[13] := ' ';
   Line[31].DFCx.ParameterSetName[14] := ' ';
   Line[31].DFCx.ParameterSetName[15] := ' ';
   Line[31].DFCx.ParameterSetName[16] := ' ';
   Line[31].DFCx.ParameterSetName[17] := ' ';
   Line[31].DFCx.ParameterSetName[18] := ' ';
   Line[31].DFCx.ParameterSetName[19] := ' ';
   Line[31].DFCx.ParameterSetName[20] := ' ';
   Line[31].DFCx.ParameterSetName[21] := ' ';
   Line[31].DFCx.ParameterSetName[22] := ' ';
   Line[31].DFCx.ParameterSetName[23] := ' ';
   Line[31].DFCx.ParameterSetName[24] := ' ';
   Line[31].DFCx.ParameterSetName[25] := ' ';
   Line[31].DFCx.ParameterSetName[26] := ' ';
   Line[31].DFCx.ParameterSetName[27] := ' ';
   Line[31].DFCx.ParameterSetName[28] := ' ';
   Line[31].DFCx.ParameterSetName[29] := ' ';
   Line[31].DFCx.ParameterSetName[30] := ' ';
   Line[32].DFCx.PelletingDieName[1] := ' ';
   Line[32].DFCx.PelletingDieName[2] := ' ';
   Line[32].DFCx.PelletingDieName[3] := ' ';
   Line[32].DFCx.PelletingDieName[4] := ' ';
   Line[32].DFCx.PelletingDieName[5] := ' ';
   Line[32].DFCx.PelletingDieName[6] := ' ';
   Line[32].DFCx.PelletingDieName[7] := ' ';
   Line[32].DFCx.PelletingDieName[8] := ' ';
   Line[32].DFCx.PelletingDieName[9] := ' ';
   Line[32].DFCx.PelletingDieName[10] := ' ';
   Line[32].DFCx.ParameterSetIdent[1] := ' ';
   Line[32].DFCx.ParameterSetIdent[2] := ' ';
   Line[32].DFCx.ParameterSetIdent[3] := ' ';
   Line[32].DFCx.ParameterSetIdent[4] := ' ';
   Line[32].DFCx.ParameterSetIdent[5] := ' ';
   Line[32].DFCx.ParameterSetIdent[6] := ' ';
   Line[32].DFCx.ParameterSetIdent[7] := ' ';
   Line[32].DFCx.ParameterSetIdent[8] := ' ';
   Line[32].DFCx.ParameterSetIdent[9] := ' ';
   Line[32].DFCx.ParameterSetIdent[10] := ' ';
   Line[32].DFCx.ParameterSetIdent[11] := ' ';
   Line[32].DFCx.ParameterSetIdent[12] := ' ';
   Line[32].DFCx.ParameterSetIdent[13] := ' ';
   Line[32].DFCx.ParameterSetIdent[14] := ' ';
   Line[32].DFCx.ParameterSetIdent[15] := ' ';
   Line[32].DFCx.ParameterSetIdent[16] := ' ';
   Line[32].DFCx.ParameterSetName[1] := ' ';
   Line[32].DFCx.ParameterSetName[2] := ' ';
   Line[32].DFCx.ParameterSetName[3] := ' ';
   Line[32].DFCx.ParameterSetName[4] := ' ';
   Line[32].DFCx.ParameterSetName[5] := ' ';
   Line[32].DFCx.ParameterSetName[6] := ' ';
   Line[32].DFCx.ParameterSetName[7] := ' ';
   Line[32].DFCx.ParameterSetName[8] := ' ';
   Line[32].DFCx.ParameterSetName[9] := ' ';
   Line[32].DFCx.ParameterSetName[10] := ' ';
   Line[32].DFCx.ParameterSetName[11] := ' ';
   Line[32].DFCx.ParameterSetName[12] := ' ';
   Line[32].DFCx.ParameterSetName[13] := ' ';
   Line[32].DFCx.ParameterSetName[14] := ' ';
   Line[32].DFCx.ParameterSetName[15] := ' ';
   Line[32].DFCx.ParameterSetName[16] := ' ';
   Line[32].DFCx.ParameterSetName[17] := ' ';
   Line[32].DFCx.ParameterSetName[18] := ' ';
   Line[32].DFCx.ParameterSetName[19] := ' ';
   Line[32].DFCx.ParameterSetName[20] := ' ';
   Line[32].DFCx.ParameterSetName[21] := ' ';
   Line[32].DFCx.ParameterSetName[22] := ' ';
   Line[32].DFCx.ParameterSetName[23] := ' ';
   Line[32].DFCx.ParameterSetName[24] := ' ';
   Line[32].DFCx.ParameterSetName[25] := ' ';
   Line[32].DFCx.ParameterSetName[26] := ' ';
   Line[32].DFCx.ParameterSetName[27] := ' ';
   Line[32].DFCx.ParameterSetName[28] := ' ';
   Line[32].DFCx.ParameterSetName[29] := ' ';
   Line[32].DFCx.ParameterSetName[30] := ' ';
END_DATA_BLOCK

DATA_BLOCK "T_FMODEMON"	// DB 4001
VERSION : 0.1
  STRUCT
   IN : BOOL ;	//Temporary placeholder variable
   PT : TIME ;
   Q : BOOL ;
   ET : TIME ;
   CTRL2_DB : WORD ;
   ET_ACT : DINT ;
   T_ACT : BOOL ;
   T_INIT_REQ : BOOL ;
   IN_FL : BOOL ;
  END_STRUCT ;	
BEGIN
END_DATA_BLOCK

